IF pActValue <> 0 AND pSetValue <> 0 AND_THEN MEMCMP(pSetValue, pActValue, Len) = 0
THEN //Skip write parameter if set and actual value are equel
	state													:= state + 1;	
	setValue												:= TRUE;
ELSE
	CoEWrite(bExecute := TRUE, nIndex := Index ,nSubIndex := SubIndex , pSrcBuf := pSetValue ,cbBufLen := Len , bCompleteAccess := CompleteAccess );
	IF NOT CoEWrite.bBusy
	THEN
		IF NOT CoEWrite.bError
		THEN
			IF pActValue <> 0 THEN MEMCPY(pActValue, pSetValue, Len); END_IF	
			state											:= state + 1;
		ELSE
			Busy											:= FALSE;
			Error											:= TRUE;
			ErrorId											:= CoEWrite.nErrId;
			ErrorText										:= CONCAT('Error write parameter in state:' , TO_STRING(state * -1));
			ErrorText										:= CONCAT(ErrorText , ' Id:');
			ErrorText										:= CONCAT(ErrorText , TO_STRING(ErrorId));
			State											:= 9999;
		END_IF
		CoEWrite(bExecute := FALSE);
		setValue											:= TRUE;
	END_IF		
END_IF
END_METHOD

END_FUNCTION_BLOCK

// ---- POUs/IO/Drives/SoE/AxDriveSoE_Ax5000CommutationCalib.TcPOU
FUNCTION_BLOCK AxDriveSoE_Ax5000CommutationCalib EXTENDS FbBase
VAR CONSTANT
	STEP_COUNT											:	INT := 1;
	P150_NAMEPLATE_TYPE									:	E_AX5000_P_0150_DigitalNamePlate := E_AX5000_P_0150_DigitalNamePlate.EAX5000_P_0150_DIGITALNAMEPLATE_BECKHOFF; //1= Digital nameplate = Beckhoff
	P150_COMMUTATION_MODE_FEEDBACK						:	UINT := 1; //1= Feedback commutation offset
	
//	P150_NO_NAMEPLATE									:	UINT := 0; //0= Digital nameplate = no nameplate
//	P150_COMMUTATION_MODE_ADJUSTABLE					:	UINT := 3; //3= Adjustable mechanical offset 
END_VAR
VAR_OUTPUT CONSTANT
{attribute 'displaymode':='binary'}
	OPTION_READ_ONLY									:	BYTE  := 2#0000_0001; //Read actual commutation offset of the motor (not stored value in drive)
{attribute 'displaymode':='binary'}
	OPTION_P98_IS_EMPTY									:	BYTE  := 2#0000_0010; //Digital nameplate not initialized, skip check if entries. Select this option for first time setup
END_VAR
VAR_INPUT
	AdsAddr												: 	AMSADDR; //Terminal AMS Net Addr.	
	Channel												:	USINT;

{attribute 'displaymode':='binary'}         			
	Options												:	BYTE  := 2#0000_0000; (* Option constants are predefined, so they can accordingly be passed symbolically to the block 
																					.0 = TRUE read only 
																					*)

	
	MaxComPosDifference									:	LREAL := 15.0; //Maximal commutation position offset (Parameter P167, result of command P166)
END_VAR
VAR_IN_OUT
	axis												: AXIS_REF;
END_VAR
VAR_OUTPUT

	P0053												: AX5000_P_0053; // Configured motor type
	P0058												: AX5000_P_0058; // Mechanical commutation offset after command P166
	P0150												: AX5000_P_0150; // Feedback type form startup list
	P0167												: AX5000_P_0167; //Motor and feedback connection check parameter
	P0098												: AX5000_P_0098_beckhoff := (	
															Id_prat_1:= 1113940843,
															Id_prat_2:= 1752131174,	
														//	Name_plate_type := , 
															Version_no:=2,
															Motor_vendor:= 0, //None
															Serial_number:= 999999); //Digital nameplate
	Offset												:	LREAL; //Scaled value

	SercosErrId											: UDINT;
END_VAR
VAR
(*  Memory *****************************************************)
	lastState											: INT := 0;

(*  Timer ******************************************************)
(*  Trigger ****************************************************)

(*  Blocks *****************************************************)
	SoECommand 											: FB_SoEExecuteCommand 	:= (Timeout := t#30s);
	SoEWritePassword 									: FB_SoEWritePassword 	:= (Password :=(strData := 'AX5000', iActualSize := 128, iMaxSize := 128), Timeout := DEFAULT_ADS_TIMEOUT);
	SoEReset											: FB_SoEReset 			:= (Timeout := DEFAULT_ADS_TIMEOUT);
	SoEWrite											: FB_SoEWrite 			:= (Timeout := T#30S);
	SoERead												: FB_SoERead 			:= (Timeout := DEFAULT_ADS_TIMEOUT);
	
(*  Error ******************************************************)
(*  Dummys *****************************************************)
	{attribute 'hide' := ''}
	i,j													: INT := 0;

END_VAR

	(*********************************************************)
	
(* state machine ********************************************************)
	rtExecute(CLK := Execute);
	CASE state OF
	0 : 
		Busy 											:= FALSE;
		
		IF NOT Execute THEN
			Done 										:= FALSE;
			Error 										:= FALSE;
			ErrorID 									:= 0;
			SercosErrId									:= 0;
		END_IF
		IF rtExecute.Q THEN
			IF axis.status.ControlLoopClosed AND NOT Options.1 THEN
				Error 									:= TRUE;
				ErrorID 								:= 19266; //xis is enabled but should not be enabled for this process.

			ELSIF AdsAddr.netId[0] = 0
			THEN
 				Error 									:= TRUE;
				ErrorID 								:= 15; //Invalid AMS net id
	
			ELSIF AdsAddr.port = 0
			THEN
				Error 									:= TRUE;
				ErrorID 								:= 24; //Invalid ADS Port
						
			ELSE
				Busy									:= TRUE;	
				Done 									:= FALSE;
				Error 									:= FALSE;
				ErrorID 								:= 0;
				SercosErrId								:= 0;	
				
				Offset									:= 0.0;
				MEMSET(ADR(P0053),0,SIZEOF(P0053));
				MEMSET(ADR(P0058),0,SIZEOF(P0058));
				MEMSET(ADR(P0150),0,SIZEOF(P0150));
				MEMSET(ADR(P0167),0,SIZEOF(P0167));
				
				SoECommand(Execute := FALSE, Axis := axis);
				SoEWrite(Execute := FALSE, Axis := axis);
				SoERead(Execute := FALSE, Axis := axis);
				SoEReset(Execute := FALSE, Axis := axis);
				SoEWritePassword(Execute := FALSE, Axis := axis);
		
					
				state									:= state + STEP_COUNT;
			END_IF
		END_IF
	
	1:	(*write drive password *)
		SoEWritePassword(
			NetId:= , 
			Execute:=TRUE , 
			Timeout:= , 
			Password:= , //See declaration 
			Axis:=axis , 
			Busy=> , 
			Error=> , 
			AdsErrId=> , 
			SercosErrId=> );
	
		IF NOT SoEWritePassword.busy
		THEN
			IF SoEWritePassword.Error
			THEN
				Busy									:= FALSE;
				Error									:= TRUE;
				ErrorId									:= SoEWritePassword.AdsErrId;
				SercosErrId								:= SoEWritePassword.SercosErrId;
				state 									:= 0;
			ELSE
				
				state									:= state + STEP_COUNT;
			END_IF		
			SoEWritePassword(Execute := FALSE, Axis := axis);
		END_IF
			
	2:	(* Reset active errors *)
		SoEReset(
			NetId:= , 
			Execute:=TRUE , 
			Timeout:= , 
			Axis:=axis , 
			Busy=> , 
			Error=> , 
			AdsErrId=> , 
			SercosErrId=> );
			
		IF NOT SoEReset.Busy
		THEN
			IF SoEReset.Error
			THEN
				Busy									:= FALSE;
				Error									:= TRUE;
				ErrorId									:= SoEReset.AdsErrId;
				SercosErrId								:= SOEReset.SercosErrId;
				state 									:= 0;
			ELSE
				
				state									:= state + STEP_COUNT;
			END_IF	
			SoEReset(Execute := FALSE, Axis := axis);	
		END_IF

	3: // read configured motor type
		SoERead(
			NetId:= , 
			Idn:=P_0_IDN+53 , // IDN P-0-0053 Configured motor type
			Element:=EC_SOE_ELEMENT_VALUE , 
			pDstBuf:=ADR(P0053) , 
			BufLen:=SIZEOF(P0053) , 
			Execute:=TRUE , 
			Timeout:= , 
			Axis:=axis , 
			Busy=> , 
			Error=> , 
			AdsErrId=> , 
			SercosErrId=> , 
			Attribute=> );
			
		IF NOT SoERead.Busy
		THEN
			IF SoERead.Error
			THEN
				Busy									:= FALSE;
				Error									:= TRUE;
				ErrorId									:= SoERead.AdsErrId;
				SercosErrId								:= SoERead.SercosErrId;
				state 									:= 0;
			ELSE		
				
				state									:= state + STEP_COUNT;
			END_IF	
			SoERead(Execute := FALSE, Axis := axis);	
		END_IF
		
	4: //Read feedback type form startup list
		SoERead(
			NetId:= , 
			Idn:=P_0_IDN+150 , 
			Element:=EC_SOE_ELEMENT_VALUE , 
			pDstBuf:=ADR(P0150) , 
			BufLen:=SIZEOF(P0150) , 
			Execute:=TRUE , 
			Timeout:= , 
			Axis:=axis , 
			Busy=> , 
			Error=> , 
			AdsErrId=> , 
			SercosErrId=> , 
			Attribute=> );
			
		IF NOT SoERead.Busy
		THEN
			IF SoERead.Error
			THEN
				Busy									:= FALSE;
				Error									:= TRUE;
				ErrorId									:= SoERead.AdsErrId;
				SercosErrId								:= SoERead.SercosErrId;
				state 									:= 0;
			ELSE				
				state									:= state + STEP_COUNT;
			END_IF		
			SoERead(Execute := FALSE, Axis := axis);
		END_IF		
		
	5: (* Reserved *****************************************************)
		state											:= state + STEP_COUNT;
		
	6: //Read nameplate to check content (must be initialized) *************************
		SoERead(
			NetId:= , 
			Idn:=P_0_IDN+98 , 
			Element:=EC_SOE_ELEMENT_VALUE , 
			pDstBuf:=ADR(P0098) , 
			BufLen:=SIZEOF(P0098) , 
			Execute:=TRUE, 
			Timeout:= , 
			Axis:=axis , 
			Busy=> , 
			Error=> , 
			AdsErrId=> , 
			SercosErrId=> , 
			Attribute=> );	
		
		IF NOT SoERead.Busy
		THEN
			IF SoERead.Error
			THEN
				Busy									:= FALSE;
				Error									:= TRUE;
				ErrorId									:= SoERead.AdsErrId;
				SercosErrId								:= SoERead.SercosErrId;
				state 									:= 0;
			ELSE
				Offset									:= TO_LREAL(P0098.Position_offset) * 0.01;
				SoERead(Execute := FALSE, Axis := axis);	
				//Check parameter of P150
				IF Options.0
				THEN //Read only
					Busy								:= FALSE;
					Done								:= TRUE;
					state 								:= 0;
					
				ELSIF Options.1
				THEN //Nameplate not active, ignore current setting
					state								:= 10;	
					
				ELSIF TO_UINT(P0150.ParameterChannel.CommutationMode0) <> P150_COMMUTATION_MODE_FEEDBACK 
				THEN
					Busy								:= FALSE;
					Error								:= TRUE;
					ErrorId								:= E_AdsErr.DEVICE_INVALIDPARM;
					SercosErrId							:= 16#F749; //Feedback parameter invalid
					state 								:= 0;	
				ELSIF P0150.ParameterChannel.DigitalNamePlate <> P150_NAMEPLATE_TYPE
				THEN
					Busy								:= FALSE;
					Error								:= TRUE;
					ErrorId								:= E_AdsErr.DEVICE_INVALIDPARM;
					SercosErrId							:= 16#F749; //Invalid nameplate
					state 								:= 0;			
			
				ELSIF P0098.Name_plate_type <> P0150.ParameterChannel.DigitalNamePlate 
				THEN
					Busy								:= FALSE;
					Error								:= TRUE;
					ErrorId								:= E_AdsErr.DEVICE_INVALIDPARM;
					SercosErrId							:= 16#F803; //Unknow nameplate
					state 								:= 0;					
				
				ELSIF P0098.Position_offset = 0.0 
				THEN
					Busy								:= FALSE;
					Error								:= TRUE;
					ErrorId								:= E_AdsErr.DEVICE_INVALIDPARM;
					SercosErrId							:= 16#F742; //Invalid commutation offset
					state 								:= 0;
						
				ELSIF P0098.Feedback_typ <> P0150.FeedbackTypeString 
				THEN
					Busy								:= FALSE;
					Error								:= TRUE;
					ErrorId								:= E_AdsErr.DEVICE_INVALIDPARM;
					SercosErrId							:= 16#F708; //Feedback type invalid
					state 								:= 0;		
				ELSIF P0098.Motor_type <> P0053.Configures_motor_type 
				THEN
					Busy								:= FALSE;
					Error								:= TRUE;
					ErrorId								:= E_AdsErr.DEVICE_INVALIDPARM;
					SercosErrId							:= 16#FD09; //Motor type invalid
					state 								:= 0;				
				ELSE
					state								:= 10;	
				END_IF	
			END_IF
		END_IF
		
	10:	// Start command P-0-0160 - calibrate commutation offset ***********************************************	
		SoECommand(
			NetId:='' , 
			Idn:=P_0_IDN+160 , //command P-0-0160 = calibrate commutation offset 
			Execute:= TRUE, 
			Timeout:= , 
			Axis:=axis , 
			Busy=> , 
			Error=> , 
			AdsErrId=> , 
			SercosErrId=> );
		
		IF NOT SoECommand.Busy
		THEN
			IF SoECommand.Error
			THEN
				Busy									:= FALSE;
				Error									:= TRUE;
				ErrorId									:= SoECommand.AdsErrId;
				SercosErrId								:= SoECommand.SercosErrId;
				state 									:= 0;
			ELSE
				state									:= state + STEP_COUNT;
			END_IF		
			SoECommand(Execute := FALSE, Axis := axis);
		END_IF
	
	11: // read mechanical commutation offset result of command P160
		SoERead(
			NetId:= , 
			Idn:=P_0_IDN+58 , // IDN P-0-0167 = parameters to check commutation and rotation direction
			Element:=EC_SOE_ELEMENT_VALUE , 
			pDstBuf:=ADR(P0058) , 
			BufLen:=SIZEOF(P0058) , 
			Execute:= TRUE , 
			Timeout:= , 
			Axis:=axis , 
			Busy=> , 
			Error=> , 
			AdsErrId=> , 
			SercosErrId=> , 
			Attribute=> );	
		
		IF NOT SoERead.Busy
		THEN
			IF SoERead.Error
			THEN
				Busy									:= FALSE;
				Error									:= TRUE;
				ErrorId									:= SoERead.AdsErrId;
				SercosErrId								:= SoERead.SercosErrId;
				state 									:= 0;
			ELSE
				//Init nameplate information - see also declaration
				P0098.Motor_type						:= P0053.Configures_motor_type;
				P0098.Feedback_typ						:= P0150.FeedbackTypeString;	
				P0098.Name_plate_type					:= P0150.ParameterChannel.DigitalNamePlate;
				P0098.Position_offset					:= P0058.Mechanical_commutation_offset;
				Offset									:= TO_LREAL(P0058.Mechanical_commutation_offset) * 0.01;		
	
				state									:= state + STEP_COUNT;
			END_IF	
			SoERead(Execute := FALSE, Axis := axis);	
		END_IF
		
	12: // Start command P-0-0166 - Motor and feedback connection check 
		SoECommand(
			NetId:='' , 
			Idn:=P_0_IDN+166 , //command P-0-0166 = motor and feedback connection check 
			Execute:= TRUE, 
			Timeout:= , 
			Axis:=axis , 
			Busy=> , 
			Error=> , 
			AdsErrId=> , 
			SercosErrId=> );
		
		IF NOT SoECommand.Busy
		THEN
			IF SoECommand.Error
			THEN
				Busy									:= FALSE;
				Error									:= TRUE;
				ErrorId									:= SoECommand.AdsErrId;
				SercosErrId								:= SoECommand.SercosErrId;
				state 									:= 0;
			ELSE
				
				state									:= state + STEP_COUNT;
			END_IF		
			SoECommand(Execute := FALSE, Axis := axis);
		END_IF
	
	13: // read P-0-0167 read connection check results
		SoERead(
			NetId:= , 
			Idn:=P_0_IDN+167 , // IDN P-0-0167 = parameters to check commutation and rotation direction
			Element:=EC_SOE_ELEMENT_VALUE , 
			pDstBuf:=ADR(P0167) , 
			BufLen:=SIZEOF(P0167) , 
			Execute:= TRUE , 
			Timeout:= , 
			Axis:=axis , 
			Busy=> , 
			Error=> , 
			AdsErrId=> , 
			SercosErrId=> , 
			Attribute=> );
				
		IF NOT SoERead.Busy
		THEN
			IF SoERead.Error
			THEN
				Busy									:= FALSE;
				Error									:= TRUE;
				ErrorId									:= SoERead.AdsErrId;
				SercosErrId								:= SoERead.SercosErrId;
				state 									:= 0;
			ELSE				
				IF P0167.EqualDirektions <> 1
					OR
					TO_LREAL(P0167.Commutation_position_difference) * 0.01 > MaxComPosDifference 
					AND TO_LREAL(P0167.Commutation_position_difference) * 0.01 < 360.0 - MaxComPosDifference
				THEN
					Busy								:= FALSE;
					Error								:= TRUE;
					ErrorId								:= E_AdsErr.DEVICE_INVALIDPARM;
					SercosErrId							:= 16#F702; //Feedback position invalid
					state 								:= 0;
				ELSE                                	
					state								:= state + STEP_COUNT;
				END_IF
			END_IF		
			SoERead(Execute := FALSE, Axis := axis);
		END_IF
		
	14:	// Write digital motor plate with commutation offset
		SoEWrite(
			NetId:= , 
			Idn:=P_0_IDN+98, // P0-0-0098 = digital motor plate 
			Element:=EC_SOE_ELEMENT_VALUE , 
			pSrcBuf:=ADR(P0098) ,
			BufLen:=SIZEOF(P0098) ,
			Execute:=TRUE,
			Timeout:= , 
			Password:= SoEWritePassword.Password, 
			Axis:=axis , 
			Busy=> , 
			Error=> , 
			AdsErrId=> , 
			SercosErrId=> );
			
		IF NOT SoEWrite.Busy
		THEN
			IF SoEWrite.Error
			THEN
				Busy									:= FALSE;
				Error									:= TRUE;
				ErrorId									:= SoEWrite.AdsErrId;
				SercosErrId								:= SoEWrite.SercosErrId;
				state 									:= 0;
			ELSE
				
				state									:= state + STEP_COUNT;
			END_IF	
			SoEWrite(Execute := FALSE, Axis := axis);	
		END_IF

	15: // Command P-0-0162 - Save digital name plate
		SoECommand(
			NetId:= , 
			Idn:=P_0_IDN+162 , //save digital name plate 
			Execute:=TRUE , 
			Timeout:= , 
			Axis:=axis , 
			Busy=> , 
			Error=> , 
			AdsErrId=> , 
			SercosErrId=> );
	
		IF NOT SoECommand.Busy
		THEN
			IF SoECommand.Error
			THEN
				Busy									:= FALSE;
				Error									:= TRUE;
				ErrorId									:= SoECommand.AdsErrId;
				SercosErrId								:= SoECommand.SercosErrId;
				state 									:= 0;
			ELSE
				
				state									:= state + STEP_COUNT;
			END_IF		
			SoECommand(Execute := FALSE, Axis := axis);
		END_IF

	16: // Write digital motor plate with commutation offset again
		SoEWrite(
			NetId:= , 
			Idn:=P_0_IDN+98 , 
			Element:=EC_SOE_ELEMENT_VALUE , 
			pSrcBuf:=ADR(P0098) ,
			BufLen:=SIZEOF(P0098) ,
			Execute:= TRUE,
			Timeout:= , 
			Password:=SoEWritePassword.Password  , 
			Axis:=axis , 
			Busy=> , 
			Error=> , 
			AdsErrId=> , 
			SercosErrId=> );
				
		IF NOT SoEWrite.Busy
		THEN
			IF SoEWrite.Error
			THEN
				Busy									:= FALSE;
				Error									:= TRUE;
				ErrorId									:= SoEWrite.AdsErrId;
				SercosErrId								:= SoEWrite.SercosErrId;
				state 									:= 0;
			ELSE
				
				state									:= state + STEP_COUNT;
			END_IF	
			SoEWrite(Execute := FALSE, Axis := axis);	
		END_IF

	17: //Start command P-0-0161 - Save commutation offset in feedback 1
		SoECommand(
			NetId:= , 
			Idn:=P_0_IDN+161 , //save commutation offset 
			Execute:=TRUE , 
			Timeout:= , 
			Axis:=axis , 
			Busy=> , 
			Error=> , 
			AdsErrId=> , 
			SercosErrId=> );
		
		IF NOT SoECommand.Busy
		THEN
			IF SoEWrite.Error
			THEN
				Busy									:= FALSE;
				Error									:= TRUE;
				ErrorId									:= SoEWrite.AdsErrId;
				SercosErrId								:= SoEWrite.SercosErrId;
				state 									:= 0;
			ELSE
				Busy									:= FALSE;
				Done									:= TRUE;
				state 									:= 0;					
			END_IF		
			SoECommand(Execute := FALSE, Axis := axis);
		END_IF
	
	ELSE
		;
	END_CASE

(* Record last state ******************************************)
IF state <> lastState AND state <> 0 AND NOT Error
THEN 
	lastState											:= state;
END_IF

(*************************************************************)

{attribute 'monitoring' := 'call'}
PROPERTY PUBLIC optP98IsEmpty : BOOL
GET
optP98IsEmpty := Options.1;
END_GET
SET
Options.1 := optP98IsEmpty;
END_SET
END_PROPERTY

{attribute 'monitoring' := 'call'}
PROPERTY PUBLIC optReadOnly : BOOL
GET
optReadOnly := Options.0;
END_GET
SET
Options.0 := optReadOnly;
END_SET
END_PROPERTY

END_FUNCTION_BLOCK

// ---- POUs/IO/Drives/SoE/AxDriveSoE_Ax5000SwitchParamSet.TcPOU
FUNCTION_BLOCK AxDriveSoE_Ax5000SwitchParamSet EXTENDS FbBase
VAR_INPUT
	rAxis													:	REFERENCE TO AXIS_REF := 0; 	// Axis Ref
	TimeOut													:	TIME := DEFAULT_ADS_TIMEOUT;	// Timeout time
	NewParamSet												:	INT;							// Value for new parameterset
END_VAR
VAR_IN_OUT	
(* important for function *)	
	AdsAddr													:	AMSADDR;						// AdsAddr of AX5000
	Channel													:	USINT;                          // Drive channel number
END_VAR
VAR_OUTPUT
	ErrorText												:	T_MaxString;					// Error Text
	ActParamSet												:	INT := -1; 						// Value of active parameter set
END_VAR
VAR
(* Memory **********************************************************)
	StartSwitchParamSet										:	INT := 0;
	
	CountError												:	USINT;
(* Timer ***********************************************************)
	TimerWait												:	TON;
	TimerTimeOut											:	TON;
	
(* Functionsblocks *************************************************)

	SoEWrite												:	FB_SoEWrite_ByDriveRef	:= (tTimeOut := DEFAULT_ADS_TIMEOUT);
	SoERead													:	FB_SoERead_ByDriveRef	:= (tTimeOut := DEFAULT_ADS_TIMEOUT);
(*******************************************************************)
END_VAR
VAR CONSTANT
	ST_IDLE													:	INT := 0;
	ST_REFRESH												:	INT := 10;
	ST_PRESELECT											:	INT := 100;
	ST_DISABLED												:	INT := 110;
	ST_RESETEXECUTE											:	INT := 120;
	ST_SETPARAM												:	INT := 130;
	ST_WAIT													:	INT := 140;
	ST_ERROR												:	INT := 998;
	ST_RESET												:	INT := 999;
	
	ERR_REFRESH												:	UDINT := 1;
	ERR_PRESELECT											:	UDINT := 2;
	ERR_TIMEOUT_DISABLED									:	UDINT := 3;
	ERR_RESETEXECUTE										:	UDINT := 4;
	ERR_EXECUTE												:	UDINT := 5;
	
	PT_WAIT_TIME											:	TIME := T#20MS;
END_VAR

(* abort function-call if the reference is invalid *****************)
	IF NOT __ISVALIDREF(rAxis) THEN
		Busy												:= NOT Error;
		Error												:= TRUE;
		ErrorId												:= 16#4B30;
		ErrorText											:= 'Referenz rAxis invalid (0)';
		RETURN;
	END_IF

(* Init drive ref **************************************************)
	IF AdsAddr.port <> SoERead.stDriveRef.nSlaveAddr
	THEN
		SoERead.stDriveRef.sNetId							:= F_CreateAmsNetId(AdsAddr.netId);
		SoERead.stDriveRef.nSlaveAddr						:= AdsAddr.port;
		SoERead.stDriveRef.nDriveNo							:= Channel;
		
		SoEWrite.stDriveRef									:= SoERead.stDriveRef;
	END_IF
(* Trigger Execute *************************************************)
	rtExecute(CLK := Execute);
	
(* switch parameter set ********************************************)
	CASE State OF
	ST_IDLE:			// wait for command
	(* Get actual parameter set after restart *)
		IF ActParamSet < 0 
		THEN
			State											:= ST_REFRESH;
	(* Start switch parameter set *)
		ELSIF rtExecute.Q
		THEN
			setNewParam(NewParamSet);
		ELSIF NOT Execute
		THEN
			Error											:= FALSE;
			Done											:= FALSE;
			Busy											:= TRUE;
			ErrorId											:= 0;
			ErrorTExt										:= '';
		END_IF
		
	ST_REFRESH: 		// Refresh ActParamSet Variable
		IF NOT SoERead.bBusy
			AND SoERead.bExecute
		THEN
			State											:= SEL(SoERead.bError, ST_IDLE, ST_ERROR);
			Done											:= State = ST_IDLE;
			Error											:= State = ST_ERROR;	
			ErrorID											:= SEL(SoERead.bError, 0, ERR_REFRESH);
			ErrorText										:= SEL(SoERead.bError, '', 'Fehler beim Aktualisieren des aktuellen Parametersatzes');
		END_IF
		
		SoERead(
			stDriveRef	:= ,  //See init for drive ref
			nIdn		:= S_0_IDN + 254,
			nElement	:= EC_SOE_ELEMENT_VALUE (* 16#40*),
			pDstBuf		:= ADR(ActParamSet),
			cbBufLen	:= SIZEOF(ActParamSet),
			bExecute	:= State = ST_REFRESH,
			tTimeout	:= ,
			bBusy		=> ,
			bError		=> ,
			iAdsErrId	=> ,
			iSercosErrId=> ,
			dwAttribute	=> );
			
		ST_PRESELECT:		// Set New param value in drive preselection
			IF NewParamSet = ActParamSet
			THEN
				State										:= ST_IDLE;
			ELSIF NOT SoEWrite.bBusy
				AND SoEWrite.bExecute
			THEN
				State										:= SEL(SoEWrite.bError, ST_DISABLED, ST_ERROR);
				ErrorID										:= SEL(SoERead.bError, 0, ERR_PRESELECT);
				ErrorText									:= SEL(SoERead.bError, '', 'Fehler beim Schreiben der Vorwahl');
			END_IF
			
			SoEWrite(
				stDriveRef	:= ,  //See init for drive ref
				nIdn		:= S_0_IDN + 217,
				nElement	:= EC_SOE_ELEMENT_VALUE (* 16#40*),
				pSrcBuf		:= ADR(NewParamSet),
				cbBufLen	:= SIZEOF(NewParamSet),
				bExecute	:= State = ST_PRESELECT,
				tTimeout	:= ,
				bBusy		=> ,
				bError		=> ,
				iAdsErrId	=> ,
				iSercosErrId=> );
				
		ST_DISABLED:		// check if axis is disabled
			TimerTimeOut(IN := NOT rAxis.Status.Disabled, PT := TimeOut);
			IF TimerTimeOut.Q THEN
				TimerTimeOut(IN := FALSE);
				State											:= ST_ERROR;
				ErrorID											:= SEL(SoERead.bError, 0, ERR_TIMEOUT_DISABLED);
				ErrorText										:= SEL(SoERead.bError, '', 'Achse ist nicht deaktiviert');
			ELSIF rAxis.Status.Disabled THEN
				TimerTimeOut(IN := FALSE);
				State											:= ST_RESETEXECUTE;
			END_IF
		
		ST_RESETEXECUTE:	// reset the execute command in drive	
			StartSwitchParamSet									:= 0;
			IF NOT SoEWrite.bBusy
				AND SoEWrite.bExecute
			THEN
				State											:= SEL(SoEWrite.bError, ST_SETPARAM, ST_ERROR);
				ErrorID											:= SEL(SoERead.bError, 0, ERR_RESETEXECUTE);
				ErrorText										:= SEL(SoERead.bError, '', 'Fehler beim Zurücksetzen des Ausführungskomamando');
			END_IF
			SoEWrite(
				stDriveRef	:= ,  //See init for drive ref
				nIdn		:= S_0_IDN + 216,
				nElement	:= EC_SOE_ELEMENT_VALUE (* 16#40*),
				pSrcBuf		:= ADR(StartSwitchParamSet),
				cbBufLen	:= SIZEOF(StartSwitchParamSet),
				bExecute	:= State = ST_RESETEXECUTE,
				tTimeout	:= ,
				bBusy		=> ,
				bError		=> ,
				iAdsErrId	=> ,
				iSercosErrId=> );		
				
		ST_SETPARAM:		// Execute switch parameter set
			StartSwitchParamSet								:= 3;
			IF NOT SoEWrite.bBusy
				AND SoEWrite.bExecute
			THEN
				State										:= SEL(SoEWrite.bError, ST_WAIT, ST_ERROR);
				ErrorID										:= SEL(SoERead.bError, 0, ERR_EXECUTE);
				ErrorText									:= SEL(SoERead.bError, '', 'Fehler beim Setzen des Ausführungskommandos');
			END_IF
			SoEWrite(
				stDriveRef	:= ,  //See init for drive ref
				nIdn		:= S_0_IDN + 216,
				nElement	:= EC_SOE_ELEMENT_VALUE (* 16#40*),
				pSrcBuf		:= ADR(StartSwitchParamSet),
				cbBufLen	:= SIZEOF(StartSwitchParamSet),
				bExecute	:= State = ST_SETPARAM,
				tTimeout	:= ,
				bBusy		=> ,
				bError		=> ,
				iAdsErrId	=> ,
				iSercosErrId=> );
				
		ST_WAIT:			// wait a short time while the drive works with the command
			TimerWait(IN := TRUE, pt := PT_WAIT_TIME);
			IF TimerWait.Q THEN
				TimerWait(IN := FALSE);
				State										:= ST_REFRESH;
			END_IF
			
		ST_ERROR:			// wait till Error is quit
			IF TRUE
			THEN
				State										:= ST_RESET;
			END_IF
			
		ST_RESET:			// Reset Error			
			State											:= ST_IDLE;
			SoEWrite(
				stDriveRef	:= ,  //See init for drive ref
				nIdn		:= S_0_IDN + 216,
				nElement	:= EC_SOE_ELEMENT_VALUE (* 16#40*),
				pSrcBuf		:= ADR(StartSwitchParamSet),
				cbBufLen	:= SIZEOF(StartSwitchParamSet),
				bExecute	:= FALSE,
				tTimeout	:= ,
				bBusy		=> ,
				bError		=> ,
				iAdsErrId	=> ,
				iSercosErrId=> );
			SoERead(
				stDriveRef	:= ,  //See init for drive ref
				nIdn		:= S_0_IDN + 254,
				nElement	:= EC_SOE_ELEMENT_VALUE (* 16#40*),
				pDstBuf		:= ADR(ActParamSet),
				cbBufLen	:= SIZEOF(ActParamSet),
				bExecute	:= FALSE,
				tTimeout	:= ,
				bBusy		=> ,
				bError		=> ,
				iAdsErrId	=> ,
				iSercosErrId=> ,
				dwAttribute	=> );
	END_CASE
	Busy													:= State <> ST_IDLE ;
(*******************************************************************)

METHOD setNewParam : BOOL	// Result = Busy
VAR_INPUT
	ParamNo					:	INT;
END_VAR

	IF ParamNo <> ActParamSet
		AND State = ST_IDLE
	THEN
		Error											:= FALSE;
		Done											:= FALSE;
		Busy											:= TRUE;
		ErrorId											:= 0;
		ErrorTExt										:= '';
		NewParamSet 									:= ParamNo;
		TimerWait(IN := FALSE);
		TimerTimeOut(IN := FALSE);
		State											:= ST_PRESELECT;
	END_IF
	
	SetNewParam											:= State <> ST_IDLE;
END_METHOD

END_FUNCTION_BLOCK

// ---- POUs/IO/EL-EP/EL1262_Base.TcPOU
FUNCTION_BLOCK EL1262_Base
VAR_INPUT
END_VAR
VAR_OUTPUT
	Input										AT %I*		:	BOOL;
{attribute 'displaymode':='binary'}
	Status										AT %I*		:	USINT;
	TimeLatchPos								AT %I*		:	T_DCTIME64;
	TimeLatchNeg								AT %I*		:	T_DCTIME64;
END_VAR
VAR
END_VAR

END_FUNCTION_BLOCK

// ---- POUs/IO/EL-EP/EL9x/EL9501.TcPOU
{attribute 'no_check'}
FUNCTION_BLOCK EL9501 EXTENDS EcSlaveInfoDataExt
VAR_INPUT
	SetVoltage					AT %Q*		:	REAL; // 0.0 - 20.0 [V]
END_VAR                 					 	
VAR_OUTPUT    
	{attribute 'displaymode':='binary'}             	
	Status						AT  %I*		:	WORD; // Terminal status (2 bytes)
          					 	
	Voltage								 	: 	AnalogInREAL ; 
	Current								 	: 	AnalogInREAL;
END_VAR                                 
VAR                                     

END_VAR

	(* EL9501 Power supply terminal	 0-20V	*)
	(****************************************)
	SUPER^();
	
(* Work objects *****************************)
	Voltage();
	Current();

(********************************************)

{attribute 'monitoring' := 'call'}
PROPERTY PUBLIC error : BOOL
GET
Error				:= Status.6 OR Voltage.Error OR Current.Error;
END_GET
END_PROPERTY

METHOD PUBLIC off : BOOL
VAR_INPUT
END_VAR
Off := CAM(SetVoltage, Voltage.Q, 0.01);
END_METHOD

{attribute 'monitoring' := 'call'}
PROPERTY PUBLIC overload : BOOL
GET
Overload 			:= Status.1;
END_GET
END_PROPERTY

{attribute 'monitoring' := 'call'}
PROPERTY PUBLIC overrange : BOOL
GET
Overrange 			:= Status.3;
END_GET
END_PROPERTY

{attribute 'monitoring' := 'call'}
PROPERTY PUBLIC underrange : BOOL
GET
Underrange 			:= Status.2;
END_GET
END_PROPERTY

{attribute 'monitoring' := 'call'}
PROPERTY PUBLIC warning : BOOL
GET
Warning 			:= Status.5;
END_GET
END_PROPERTY

END_FUNCTION_BLOCK

// ---- POUs/IO/_EcSlaveInfoDataIO/EcSlaveInfoDataExt.TcPOU
{attribute 'no_check'}
{attribute 'reflection'} 
FUNCTION_BLOCK EcSlaveInfoDataExt Extends EcSlaveInfoData
VAR_INPUT
END_VAR                         					
VAR_OUTPUT                      					
	AmsNetIdStr												: T_AmsNetId; //AMS NetID string
	EcMasterDevId									AT %I*	: UINT; 	// Link to EtherCAT Master "DevId" under InfoData 
	DevName													:	STRING(30) := ''; //Slave device name as give in IO tree				
	{attribute 'instance-path'} 
    {attribute 'noinit'} 
    InstancePath 											: STRING; 	
END_VAR
VAR
	IOF_GetBoxNameByAddr									:	IOF_GetBoxNameByAddr := (NETID := '', TMOUT := DEFAULT_ADS_TIMEOUT);
	_Init_													: BOOL;
END_VAR

(* Get device name by address and master device id								*)
(********************************************************************************)

(* Get name *********************************************************************)
IF NOT _Init_
THEN 	
	IF NOT IOF_GetBoxNameByAddr.START
	THEN
		IF AdsAddr.port = 0 
		THEN
			adsLogError('AdsAddr.port invalid: %s', InstancePath);
		END_IF
		IF EcMasterDevId = 0 
		THEN
			adsLogError('EcMasterDevId invalid: %s', InstancePath);
		END_IF
			
		IF AdsAddr.port > 0 AND EcMasterDevId > 0
		THEN
			IOF_GetBoxNameByAddr.START						:= TRUE;
			AmsNetIdStr										:= F_CreateAmsNetId(nIds := AdsAddr.netId);
		END_IF		
	END_IF
	
	IOF_GetBoxNameByAddr(
		NETID		:=  , (* Local *)
		DEVICEID	:= TO_UDINT(EcMasterDevId) ,
		BOXADDR		:= AdsAddr.port ,
		START		:= ,
		TMOUT		:= ,
		BOXNAME		=> DevName);
	IF NOT IOF_GetBoxNameByAddr.BUSY 
	THEN
		IF IOF_GetBoxNameByAddr.ERR 
		THEN
			adsLogError(CONCAT(CONCAT('ADS Error ', DWORD_TO_HEXSTR(IOF_GetBoxNameByAddr.ERRID,4,FALSE)),' reading BoxName of EtherCAT Device: %s'), InstancePath);
		END_IF
		IOF_GetBoxNameByAddr(START:= FALSE);
		_Init_												:= TRUE;
	END_IF
END_IF
(********************************************************************************)

END_FUNCTION_BLOCK

// ---- POUs/IO/EL-EP/EL3356.TcPOU
{attribute 'no_check'}
//EL3356 load cell analysis (resistor bridge) process image
//Mode of operation = Standard (Real or INT32)
FUNCTION_BLOCK EL3356 EXTENDS EcSlaveInfoDataExt
VAR_INPUT
//RMB Control
	StartCalib										AT  %Q* : 	BOOL; 
	DisableCalib									AT  %Q* : 	BOOL;
	InputFreeze										AT  %Q* : 	BOOL;
	SampleMode										AT  %Q* : 	BOOL; //1=High speed and low latency / only on EL3356-0010
	Tara											AT  %Q* : 	BOOL;				
END_VAR                     			    					
VAR_OUTPUT                      					
//RMB Status
	Overrange										AT  %I*	:	BOOL;
	DataInvalid										AT  %I*	:	BOOL;
	Error											AT  %I*	:	BOOL;
	CalibInProgress									AT  %I*	:	BOOL;
	SteadyState										AT  %I*	:	BOOL;
	SyncError										AT  %I*	:	BOOL;
	TxPDOToggle										AT  %I* : 	BOOL;
	
//RMB Value
	InReal											AT  %I* : 	REAL; //RMP Value Real 32		
	InInt32											AT  %I* : 	DINT; //RMB Value INT32
END_VAR
VAR
END_VAR

(* EL3356 IOs											             	 		*)
(********************************************************************************)

(* ******************************************************************************)
	Super^();
(********************************************************************************)

{attribute 'monitoring' := 'call'}
PROPERTY PUBLIC inError : BOOL
GET
inError													:= Error OR SyncError OR WcState OR InfoDataState <> Tc2_EtherCAT.EC_DEVICE_STATE_OP;
END_GET
END_PROPERTY

{attribute 'monitoring' := 'call'}
PROPERTY PUBLIC Q : LREAL
GET
IF InInt32 <> 0
THEN
	Q 														:= TO_LREAL(InInt32);
ELSE
	Q 														:= TO_LREAL(InReal);
END_IF
END_GET
END_PROPERTY

{attribute 'monitoring' := 'call'}
PROPERTY Q_GramToNewton : LREAL
GET
Q_GramToNewton := GF_TO_N(Q);
END_GET
END_PROPERTY

{attribute 'monitoring' := 'call'}
PROPERTY Q_NewtonToGram : LREAL
GET
Q_NewtonToGram := N_TO_GF(Q);
END_GET
END_PROPERTY

END_FUNCTION_BLOCK

// ---- POUs/_Miscellaneous/Conversions/GF_TO_N.TcPOU
{attribute 'no_check'}
//Gram-force to newton
FUNCTION GF_TO_N : LREAL
VAR_INPUT
	GF				:	LREAL;
END_VAR
VAR
END_VAR
(*
Gram-force to newton (gf to N):
Fn = Fgf ×0.00980665
Example:
If gf = 156 then N = 1.5298374N

Newton to gram-force (N to gf):
Fgf = Fn / 0.00980665
*)

GF_TO_N := GF * 0.00980664999999998 ;

END_FUNCTION

// ---- POUs/_Miscellaneous/Conversions/N_TO_GF.TcPOU
{attribute 'no_check'}
//Newton to Gram-force
FUNCTION N_TO_GF : LREAL
VAR_INPUT
	FN				:	LREAL;
END_VAR
VAR
END_VAR
(*
Gram-force to newton (gf to N):
Fn = Fgf ×0.00980665
Example:
If gf = 156 then N = 1.5298374N

Newton to gram-force (N to gf):
Fgf = Fn / 0.00980665
*)

N_TO_GF := FN / 0.00980664999999998;

END_FUNCTION

// ---- POUs/IO/EL-EP/EP92xxPwrBox/EP9214_CHANNEL.TcPOU
{attribute 'no_check'}
FUNCTION_BLOCK EP9214_CHANNEL
VAR_INPUT
	EnableUs									AT  %Q* 	: 	BOOL := TRUE; 	//switches system voltage on with a rising edge
	EnableUp									AT  %Q* 	: 	BOOL := TRUE; 	//switches peripheral voltage on with a rising edge
	ResetTrigUs	                                AT  %Q* 	: 	BOOL := FALSE;  //resets system voltage with a rising edge                    
	ResetTrigUp                                 AT  %Q* 	: 	BOOL := FALSE;	//resets peripheral voltage with a rising edge                                                                                           
END_VAR     								                          
VAR_OUTPUT  								                          
	ErrorUs										AT  %I* 	: 	BOOL := FALSE;	//TRUE when system voltage error occurs 
	ErrorUp										AT  %I* 	: 	BOOL := FALSE; 	//TRUE when peripheral voltage error occurs 
	WarningUs									AT  %I* 	: 	BOOL := FALSE; 	//TRUE when system voltage warning occurs 
	WarningUp									AT  %I* 	: 	BOOL := FALSE; 	//TRUE when peripheral voltage warning occurs 
	StatusUs									AT  %I* 	: 	BOOL := FALSE; 	//TRUE when system voltage is on
	StatusUp									AT  %I* 	: 	BOOL := FALSE; 	//TRUE when peripheral voltage is on 
	ChannelError								AT  %I* 	: 	BOOL := FALSE; 	//TRUE when channel error occurs 
	SyncError									AT  %I* 	: 	BOOL := FALSE; 	//TRUE when synchronization error occurs 
	TxPDOState									AT  %I* 	: 	BOOL := FALSE; 
	TxPDOToggle									AT  %I* 	: 	BOOL := FALSE; 
END_VAR     								
VAR
END_VAR

;

END_FUNCTION_BLOCK

// ---- POUs/IO/Fuse.TcPOU
{attribute 'no_check'}
//Fuse/Circuit breaker 
FUNCTION_BLOCK Fuse
VAR_INPUT
	Force													:	BOOL := FALSE;	//simulates Input
	Invert													:	BOOL := FALSE; 	//inverts the Hardware Input
	ResetTrig												:	BOOL := TRUE;	//Resets error with rising edge 
END_VAR     								
VAR_OUTPUT  								
	Q														:	BOOL;			//output
	Event													:	BOOL;			//TRUE when state is abnormal and error is not reset 
	In											AT  %I* 	: 	BOOL := TRUE;	//Hardware Input
END_VAR     								
VAR
END_VAR

(* signallocked Input-FB (MSS,Sicherung)				*)
(********************************************************)

(************************************)
IF NOT (In OR Force) XOR Invert
THEN
	Event													:= TRUE;
	Q														:= Invert;
ELSIF Event                         						
THEN                                						
	Event 													:= NOT ResetTrig;
ELSE                                						
	Q														:= Not Invert;
END_IF

(************************************)

METHOD PUBLIC reset : BOOL
VAR_INPUT
END_VAR
Event := FALSE;
reset := TRUE;
END_METHOD

END_FUNCTION_BLOCK

// ---- POUs/IO/InOut.TcPOU
{attribute 'no_check'}
FUNCTION_BLOCK InOut 
VAR_INPUT
	Q												AT  %Q*	:	BOOL; //Link to hardware output
END_VAR             								
VAR_OUTPUT          								
	In												AT  %I*	:	BOOL; //Link to hardware input
END_VAR
VAR
END_VAR

;

END_FUNCTION_BLOCK

// ---- POUs/IO/Motors/IOMotor.TcPOU
{attribute 'no_check'}
FUNCTION_BLOCK IOMotor IMPLEMENTS I_ActuatorOnOff
VAR_INPUT
	ResetTrig												:	BOOL := TRUE; //Confirm error
	start													:	BOOL;
	Feed													:	BOOL;
	ProtSwitchOK											: 	FUSE;
END_VAR                 							
VAR_OUTPUT
{attribute 'displaymode':='binary'}
	Status													:	BYTE;              							
	Q_Contactor										AT  %Q* :	BOOL; //Hardware output for main contactor to start motor	
	Busy													:	BOOL;
	Error													:	BOOL;
END_VAR                 							
VAR (* IO Internal *)   							

                        	
END_VAR                 	
VAR                     	
END_VAR

(* Com Motor IO 					 		V2.2		*)
(********************************************************)

(* Protection Switch *****************************************)
	IF ResetTrig THEN reset(); END_IF

	ProtSwitchOK();

(* Enable ****************************************************)
	IF Start THEN
		switchOn();
	ELSE
		switchOff();
	END_IF
	
(* HMI status *********************************************)
	_writeStatus();
	
(********************************************************)

METHOD PROTECTED _writeStatus : BOOL
VAR_INPUT
END_VAR
	
(* HmiStatus **************************************************)
	Status.0												:= NOT Q_Contactor;
	Status.1												:= Q_Contactor;
	Status.2												:= FALSE;
	Status.3												:= FALSE;
	Status.4												:= FALSE;
	Status.5												:= Feed ;
	Status.6												:= NOT Error;
	Status.7												:= Error;

	(* Result *)
	_writeStatus											:= TRUE;
    												
(**************************************************************)
END_METHOD

METHOD enable : BOOL //Result value = successful execution of desired action 
VAR_INPUT
	IN							:	BOOL; //TRUE = Enable Pos/FWD/Up/Open/Left/Work FALSE = Opposite
END_VAR
IF in
THEN
	enable := switchOn();
ELSE
	enable := switchOff();
END_IF
END_METHOD

{attribute 'monitoring' := 'call'}
PROPERTY public inError : bool
GET
inError := Error;
END_GET
END_PROPERTY

{attribute 'monitoring' := 'call'}
PROPERTY public isBusy : bool
GET
isBusy := Busy;
END_GET
END_PROPERTY

{attribute 'monitoring' := 'call'}
PROPERTY public isOff : BOOL
GET
isOff := not Q_Contactor;
END_GET
END_PROPERTY

{attribute 'monitoring' := 'call'}
PROPERTY public isOn : BOOL
GET
isOn := Q_Contactor;
END_GET
END_PROPERTY

{attribute 'monitoring' := 'call'}
PROPERTY noFeed : BOOL
GET
noFeed := NOT Feed;
END_GET
END_PROPERTY

{attribute 'monitoring' := 'call'}
PROPERTY ok : bool
GET
ok := isBusy;
END_GET
END_PROPERTY

METHOD PUBLIC reset : bool
VAR_INPUT
END_VAR
Error									:= FALSE;
reset									:= ProtSwitchOK.reset();
END_METHOD

METHOD public switchOff : BOOL  //True if motor is switched off
VAR_INPUT
END_VAR
Start														:= FALSE;
Q_Contactor 												:= FALSE;
Busy														:= FALSE;
Error														:= NOT ProtSwitchOK.Q;
switchOff													:= TRUE;
END_METHOD

METHOD public switchOn : BOOL  //True if motor is switched on
VAR_INPUT
END_VAR
Start														:= TRUE;
Q_Contactor		 											:= ProtSwitchOK.Q AND Feed;
switchOn													:= Q_Contactor;
Busy														:= switchOn;
Error														:= NOT ProtSwitchOK.Q;
END_METHOD

END_FUNCTION_BLOCK

// ---- POUs/IpcDiag/MDP/InfoModuls/MDP_Mainboard.TcPOU
{attribute 'no_check'}
FUNCTION_BLOCK MDP_Mainboard  EXTENDS FbBase
VAR_OUTPUT CONSTANT
	MIN_VOLTAGE												:	INT := 1;
	MAX_VOLTAGE												:	INT := 20;

(* Voltage Location *)
 	VLOC_UNKNOWN											:	INT := 0;
	VLOC_OTHER												:	INT := 1;
 	VLOC_PROCESSOR											:	INT := 2;
 	VLOC_DISK												:	INT := 3;
 	VLOC_SYSTEM_MANAGEMENT_MODULE							:	INT := 4;
 	VLOC_MOTHERBOARD										:	INT := 5;
 	VLOC_MEMORY_MODULE										:	INT := 6;
 	VLOC_POWER_SUPPLY										:	INT := 7;
 	VLOC_ADDIN_CARD											:	INT := 8;
 	VLOC_FRONT_PANEL_BOARD									:	INT := 9;
 	VLOC_BACK_PANEL_BOARD									:	INT := 10;
 	VLOC_PERIPHERIE											:	INT := 11;
 	VLOC_CHASSIS											:	INT := 12;
 	VLOC_BATTERY											:	INT := 13;
 	VLOC_UPS												:	INT := 14;
	VLOC_GRAFFIC_BOARD										:	INT := 15;
 	VLOC_SUPERIO											:	INT := 16;
	VLOC_CHIPSET											:	INT := 17;
END_VAR                             						
VAR_INPUT                           						
	AmsNetId												: 	T_AmsNetId := '';				//AmsNetId as text
	Timeout													:	TIME := DEFAULT_ADS_TIMEOUT;	//Ads timeout
END_VAR
VAR_OUTPUT
	MB_Type													:	STRING(20);	//Type of Mainboard
	SerielNo												:	STRING(20);	//Serial number of Mainboard
	ProdDate												:	STRING(20);	//Production date of Mainboard
	BootCount												:	UDINT;		//total number of boots
	OpTime													:	UDINT; 		//Operating Time
	MinBoardTemp											:	DINT;		//minimum board temperature
	MaxBoardTemp											:	DINT;		//maximum board temperature
	MinInputVolt											:	DINT;		//minimum board input voltage
	MaxInputVolt											:	DINT;		//maximum board input voltage
	MB_Temp													:	INT;		//current board temperature
	IPC_SerielNo											:	STRING(20);	//industrial PC serial number
                        									
	VoltLocation											:  	ARRAY[MIN_VOLTAGE..MAX_VOLTAGE] OF INT;	//voltage location
	VoltageValue											:	ARRAY[MIN_VOLTAGE..MAX_VOLTAGE] OF INT;	//voltage value
	VoltageNominal											:	ARRAY[MIN_VOLTAGE..MAX_VOLTAGE] OF INT;	//nominal voltage
	VoltCount												:	INT; 		//number of measuring points
	ErrorGrp												:	E_MDP_ErrGroup := eMDP_Err_NoError;

END_VAR                 									
VAR                     									
	idx														:	INT := 1;
	MDP_ScanModules											:	FB_MDP_ScanModules := ( nModuleType 	:= eMDP_ModT_Mainboard , iModIdx		:= 0);
	MDP_Read												: 	FB_MDP_Read;
	SplitErrorId											:	FB_MDP_SplitErrorID;
	DstBuf													:	ARRAY[0..21] OF BYTE;
END_VAR

(* Read Mainboard Information 				V1.0	*)
(****************************************************)

(* Start Read *******************************************************)
	IF Execute
		AND state = 0
	THEN
		MB_Type												:= '';
		SerielNo											:= '';
		ProdDate											:= '';
		BootCount											:= 0;
		OpTime												:= 0;
		MinBoardTemp										:= 0;
		MaxBoardTemp										:= 0;
		MinInputVolt										:= 0;
		MaxInputVolt										:= 0;
		MB_Temp												:= 0;
		MEMSET(ADR(VoltLocation),0,SIZEOF(VoltLocation));
		MEMSET(ADR(VoltageValue),0,SIZEOF(VoltageValue));
		MEMSET(ADR(VoltageNominal),0,SIZEOF(VoltageNominal));
		VoltCount											:= 0;

		Busy												:= TRUE;
		Done												:= FALSE;
		Error												:= FALSE;
		ErrorId												:= 0;
		ErrorGrp											:= eMDP_Err_NoError;
		MDP_Read(bExecute := FALSE);
		MDP_ScanModules(
			bExecute			:= FALSE,
			nModuleType			:= eMDP_ModT_Mainboard,
			iModIdx				:= 0,
			tTimeout			:= timeout,
			sAmsNetId			:= AmsNetId,
			bBusy				=> ,
			bError				=> ,
			nErrID				=> ,
			nDynModuleId		=> ,
			iModuleTypeCount	=> ,
			iModuleCount		=> );

		MDP_ScanModules(bExecute:= TRUE);	
		state												:= 1;
		
	ELSIF NOT Execute
		AND State = 99
	THEN
		state												:= 0;
		Busy												:= FALSE;
		Done												:= FALSE;
		Error												:= FALSE;
		ErrorId												:= 0;
		ErrorGrp											:= eMDP_Err_NoError;
	END_IF


	CASE state OF
	0:
		;

	1:
		MDP_ScanModules();
		IF NOT MDP_ScanModules.bBusy
		THEN
			IF MDP_ScanModules.bError
			THEN
				Busy										:= FALSE;
				Error										:= TRUE;
				SplitErrorId(
					nErrID		:= MDP_ScanModules.nErrID,
					eErrGroup	=> ErrorGrp ,
					nErrCode	=> ErrorId);
				state										:= 99;
				MDP_ScanModules(bExecute := FALSE);
			ELSE
				MDP_Read(bExecute := FALSE);
				MDP_Read.stMDP_DynAddr.nArea				:= 16#8;
				MDP_Read.stMDP_DynAddr.nModuleId			:= MDP_ScanModules.nDynModuleId;
				MDP_Read.stMDP_DynAddr.nTableId				:= 1;
				MDP_Read.stMDP_DynAddr.nSubIdx				:= 0;
				idx											:= 1;
				state										:= 2;
			END_IF                                  		

		END_IF

	2:
		MDP_Read( pDstBuf	:= ADR(DstBuf), cbDstBufLen := SIZEOF(DstBuf));
		IF NOT MDP_Read.bBusy
		THEN
			IF MDP_Read.bError AND MDP_Read.bExecute
			THEN
				Busy										:= FALSE;
				Error										:= TRUE;
				SplitErrorId(
					nErrID		:= MDP_Read.nErrID,
					eErrGroup	=> ErrorGrp ,
					nErrCode	=> ErrorId);
				state										:= 99;
				MDP_Read(bExecute := FALSE);
			ELSE
				MDP_Read(bExecute := FALSE);
				CASE MDP_Read.stMDP_DynAddr.nTableId OF
				1:
					CASE MDP_Read.stMDP_DynAddr.nSubIdx OF
					0:
						MDP_Read.stMDP_DynAddr.nSubIdx		:= 1;

					1:
						MEMCPY(ADR(MB_Type), ADR(DstBuf), MIN(MDP_Read.nCount, SIZEOF(MB_Type)) );
						MDP_Read.stMDP_DynAddr.nSubIdx		:= 2;

					2:
						MEMCPY(ADR(SerielNo), ADR(DstBuf), MIN(MDP_Read.nCount, SIZEOF(SerielNo)) );
						MDP_Read.stMDP_DynAddr.nSubIdx		:= 3;

					3:
						MEMCPY(ADR(ProdDate), ADR(DstBuf), MIN(MDP_Read.nCount, SIZEOF(ProdDate)) );
						MDP_Read.stMDP_DynAddr.nSubIdx		:= 4;

					4:
						MEMCPY(ADR(BootCount), ADR(DstBuf), SIZEOF(BootCount));
						MDP_Read.stMDP_DynAddr.nSubIdx		:= 5;

					5:
						MEMCPY(ADR(OpTime), ADR(DstBuf), SIZEOF(OpTime));
						MDP_Read.stMDP_DynAddr.nSubIdx		:= 6;

					6:
						MEMCPY(ADR(MinBoardTemp), ADR(DstBuf), SIZEOF(MinBoardTemp));
						MDP_Read.stMDP_DynAddr.nSubIdx		:= 7;

					7:
						MEMCPY(ADR(MaxBoardTemp), ADR(DstBuf), SIZEOF(MaxBoardTemp));
						MDP_Read.stMDP_DynAddr.nSubIdx		:= 8;

					8:
						MEMCPY(ADR(MinInputVolt), ADR(DstBuf), SIZEOF(MinInputVolt));
						MDP_Read.stMDP_DynAddr.nSubIdx		:= 9;

					9:
						MEMCPY(ADR(MaxInputVolt), ADR(DstBuf), SIZEOF(MaxInputVolt));
						MDP_Read.stMDP_DynAddr.nSubIdx		:= 10;

					10:
						MEMCPY(ADR(MB_Temp), ADR(DstBuf), SIZEOF(MB_Temp));
						MDP_Read.stMDP_DynAddr.nSubIdx		:= 0;
						MDP_Read.stMDP_DynAddr.nTableId		:= 4;
					END_CASE

				4:
					CASE MDP_Read.stMDP_DynAddr.nSubIdx OF
					0:
						MEMCPY(ADR(VoltCount), ADR(DstBuf), SIZEOF(VoltCount) );
						IF VoltCount > 0 THEN
							MDP_Read.stMDP_DynAddr.nSubIdx	:= 1;
						ELSE						
							state							:= 3;
						END_IF

					1..255:
						MEMCPY(ADR(VoltLocation[MDP_Read.stMDP_DynAddr.nSubIdx]), ADR(DstBuf), SIZEOF(VoltLocation[MIN_VOLTAGE]));
						MDP_Read.stMDP_DynAddr.nSubIdx	:= MDP_Read.stMDP_DynAddr.nSubIdx + 1;
						
						IF MDP_Read.stMDP_DynAddr.nSubIdx > VoltCount
						THEN
							MDP_Read.stMDP_DynAddr.nSubIdx	:= 1;
							MDP_Read.stMDP_DynAddr.nTableId	:= 5;
						END_IF
					END_CASE

				5:
					CASE MDP_Read.stMDP_DynAddr.nSubIdx OF
					1..255:
						MEMCPY(ADR(VoltageValue[MDP_Read.stMDP_DynAddr.nSubIdx]), ADR(DstBuf), SIZEOF(VoltageValue[MIN_VOLTAGE]));
						MDP_Read.stMDP_DynAddr.nSubIdx	:= MDP_Read.stMDP_DynAddr.nSubIdx + 1;
						
						IF MDP_Read.stMDP_DynAddr.nSubIdx > VoltCount
						THEN
							MDP_Read.stMDP_DynAddr.nSubIdx	:= 1;
							MDP_Read.stMDP_DynAddr.nTableId	:= 6;
						END_IF
					END_CASE

				6:
					CASE MDP_Read.stMDP_DynAddr.nSubIdx OF
					1..255:
						MEMCPY(ADR(VoltageNominal[MDP_Read.stMDP_DynAddr.nSubIdx]), ADR(DstBuf), SIZEOF(VoltageNominal[MIN_VOLTAGE]));
						MDP_Read.stMDP_DynAddr.nSubIdx	:= MDP_Read.stMDP_DynAddr.nSubIdx + 1;
						
						IF MDP_Read.stMDP_DynAddr.nSubIdx > VoltCount
						THEN
							state							:= 3;
						END_IF
					END_CASE
				END_CASE

				MDP_Read(
					stMDP_DynAddr	:= ,		(* address to request subindex Count of AdressList *)
					pDstBuf			:= ADR(DstBuf),
					cbDstBufLen		:= SIZEOF(DstBuf),
					bExecute		:= NOT MDP_Read.bBusy AND state = 2,
					tTimeout		:= Timeout,
					sAmsNetId		:= AmsNetId,
					bBusy			=> ,
					bError			=> ,
					nErrId			=> );
			END_IF
		END_IF

	3: //Start lesen der IPC Seriennummer 
		MDP_Read.stMDP_DynAddr.nArea						:= INT_TO_BYTE(eMDP_Area_DeviceArea);
		MDP_Read.stMDP_DynAddr.nModuleId					:= 16#9F;
		MDP_Read.stMDP_DynAddr.nTableId						:= 16#00;
		MDP_Read.stMDP_DynAddr.nSubIdx						:= 16#00;
		
		MDP_Read(
			stMDP_DynAddr	:= ,		(* address to request subindex Count of AdressList *)
			pDstBuf			:= ADR(IPC_SerielNo),
			cbDstBufLen		:= SIZEOF(IPC_SerielNo),
			bExecute		:= NOT MDP_Read.bBusy,
			tTimeout		:= Timeout,
			sAmsNetId		:= AmsNetId,
			bBusy			=> ,
			bError			=> ,
			nErrId			=> );	
			
		state												:= 4;	
	
	4:
		MDP_Read( pDstBuf	:= ADR(IPC_SerielNo), cbDstBufLen := SIZEOF(IPC_SerielNo));
		IF NOT MDP_Read.bBusy
		THEN
			IF MDP_Read.bError AND MDP_Read.bExecute
			THEN
				Busy										:= FALSE;
				Error										:= TRUE;
				SplitErrorId(
					nErrID		:= MDP_Read.nErrID,
					eErrGroup	=> ErrorGrp ,
					nErrCode	=> ErrorId);
				state										:= 99;	
			ELSE			                        		
				Busy										:= FALSE;
				Done										:= TRUE;
				state										:= 99;
			END_IF
			MDP_Read(bExecute := FALSE);
			
		END_IF

	99: ;

	ELSE
		;
	END_CASE


	(* reset state for next start *)
	IF NOT Execute
		AND state = 99
	THEN
		state												:= 0;
	END_IF

(****************************************************************************************************)

END_FUNCTION_BLOCK

// ---- POUs/IpcDiag/MDP/InfoModuls/MDP_ReadModulList.TcPOU
{attribute 'no_check'}
FUNCTION_BLOCK MDP_ReadModulList EXTENDS FbBase
VAR_INPUT
	AmsNetId												: 	T_AmsNetId := '';	//AmsNetId as text
	Timeout													:	TIME := DEFAULT_ADS_TIMEOUT;	//Ads timeout
END_VAR                     								
VAR_OUTPUT                  								
	ModulCount												:	USINT;	//number of modules
	ModulType												:	ARRAY[0..255] OF E_MDP_ModuleType; //Index = Modul ID
	ErrorGrp												:	E_MDP_ErrGroup := eMDP_Err_NoError;
END_VAR                     								
VAR                         								
	MDP_Read												: 	FB_MDP_Read		:= (stMDP_DynAddr := (nArea := INT_TO_BYTE(eMDP_Area_DeviceArea), nModuleId := 16#02, nTableId := 16#00, nFlag := 16#00, nSubIdx := 16#00));
	SplitErrorId											:	FB_MDP_SplitErrorID;
	dwData													:	ARRAY [1..2] OF WORD;
END_VAR

(* Read list ob available moduls			V1.0	*)
(****************************************************)

(* Start read ************************************************)
	IF Execute
		AND state = 0
	THEN
		IF FALSE
		THEN (* Modultypen Liste *)
			MDP_Read.stMDP_DynAddr.nModuleId				:= 16#01;
		ELSE (* Modul ID Liste *)               			
			MDP_Read.stMDP_DynAddr.nModuleId				:= 16#02;
		END_IF                                  			
		MDP_Read.stMDP_DynAddr.nSubIdx						:= 0;
		MEMSET(ADR(ModulType),0,SIZEOF(ModulType));
		ModulCount											:= 0;
		Busy												:= TRUE;
		Done												:= FALSE;
		Error												:= FALSE;
		ErrorId												:= 0;
		ErrorGrp											:= eMDP_Err_NoError;
		
		MDP_Read(
			stMDP_DynAddr	:= ,		(* address to request subindex Count of AdressList *)
			pDstBuf			:= ADR(dwData),
			cbDstBufLen		:= SIZEOF(dwData),
			bExecute		:= FALSE,
			tTimeout		:= Timeout,
			sAmsNetId		:= AmsNetId,
			bBusy			=> ,
			bError			=> ,
			nErrId			=> );

		MDP_Read(bExecute	:= TRUE);
		state												:= 1;
	ELSIF NOT Execute
		AND State = 99
	THEN
		state												:= 0;
		Busy												:= FALSE;
		Done												:= FALSE;
		Error												:= FALSE;
		ErrorId												:= 0;
		ErrorGrp											:= eMDP_Err_NoError;
	END_IF


	CASE state OF
	0:
		;
	1:
		MDP_Read(pDstBuf := ADR(dwData), cbDstBufLen := SIZEOF(dwData));
		IF NOT MDP_Read.bBusy
		THEN
			IF MDP_Read.bError AND MDP_Read.bExecute
			THEN
				Busy										:= FALSE;
				Error										:= TRUE;
				SplitErrorId(
					nErrID		:= MDP_Read.nErrID,
					eErrGroup	=> ErrorGrp ,
					nErrCode	=> ErrorId);
				state										:= 99;
				MDP_Read(bExecute := FALSE);
			ELSE
				IF ModulCount = 0
				THEN (* Init Modul count *)
					ModulCount								:= WORD_TO_USINT(dwData[1]);
				ELSIF MDP_Read.stMDP_DynAddr.nSubIdx > 0
				THEN (* copy emlement dat					a *)
					ModulType[MDP_Read.stMDP_DynAddr.nSubIdx - 1] :=  dwData[2];					
				END_IF
				MDP_Read(bExecute := FALSE);
				MDP_Read.stMDP_DynAddr.nSubIdx:= MDP_Read.stMDP_DynAddr.nSubIdx + 1;
				IF MDP_Read.stMDP_DynAddr.nSubIdx > ModulCount
					OR MDP_Read.stMDP_DynAddr.nSubIdx > 255
				THEN
					Busy									:= FALSE;
					Done									:= TRUE;
					state									:= 99;
				ELSE
					MDP_Read(bExecute := TRUE,	pDstBuf	:= ADR(dwData), cbDstBufLen := SIZEOF(dwData));
				END_IF
			END_IF

		END_IF

	99: ;

	ELSE
		;
	END_CASE

	(* reset state for next start *)
	IF NOT Execute
		AND state = 99
	THEN
		state												:= 0;
	END_IF

(****************************************************************************************************)

END_FUNCTION_BLOCK

// ---- POUs/IpcDiag/MDP/InfoModuls/MDP_UPS.TcPOU
{attribute 'no_check'}
FUNCTION_BLOCK MDP_UPS EXTENDS FbBase
VAR_OUTPUT CONSTANT
(* Battery Power Status *)
	PS_UNKNOWN												:	INT := 0;
	PS_ONLINE												:	INT := 1;
	PS_ONBATTERIES											:	INT := 2;
	                    									
(* Com Status *)        									
	CS_UNKNOWN												:	INT := 0;
	CS_OK													:	INT := 1;
	CS_ERROR												:	INT := 2;

(* Battery Power Status *)
	BS_UNKNOWN												:	INT := 0;
	BS_OK													:	INT := 1;
	BS_CHANGE_BATTERY										:	INT := 2;
	
END_VAR
VAR_INPUT
	AmsNetId												: 	T_AmsNetId := '';	//AmsNetId
	Timeout													:	TIME := DEFAULT_ADS_TIMEOUT;	//Ads timeout
END_VAR
VAR_OUTPUT
(* UPS Data *)              								
	Model													:	STRING(30);	//model name
	VendorName												:	STRING(30);	//vendor name
	PowerStatus												:	INT := PS_UNKNOWN;
	ComStatus												:	INT := CS_UNKNOWN;
	BatteryStatus											:	INT := BS_UNKNOWN;
	BatteryCapacity											:	USINT; 		//in %
	BatteryRuntime											:	UDINT; 		//in sec
	PersPowerFailCounter									:	BOOL;		//TRUE when persistent power fail counter is activated
	PowerFailCounter										:	UDINT;		//number of power fails
	FanError												:	BOOL;		//Fan has error
	NoBattery												:	BOOL;		//No battery connected
	ErrorGrp												:	E_MDP_ErrGroup := eMDP_Err_NoError;

END_VAR                     								
VAR                         								
	idx														:	INT := 1;
	MDP_ScanModules											:	FB_MDP_ScanModules := ( nModuleType 	:= eMDP_ModT_UPS , iModIdx		:= 0);
	MDP_Read												: 	FB_MDP_Read;
	SplitErrorId											:	FB_MDP_SplitErrorID;
	DstBuf													:	ARRAY[0..31] OF BYTE;
END_VAR

	(* Read UPS Information 							V1.0	*)
	(***************************************************)

(* Start Read *******************************************************)
	IF Execute
		AND state = 0
	THEN
		Model												:= '';
		VendorName											:= '';
		PowerStatus											:= PS_UNKNOWN;
		ComStatus											:=	CS_UNKNOWN;
		BatteryStatus										:=	BS_UNKNOWN;
		BatteryCapacity										:= 0;
		BatteryRuntime										:= 0;
		PowerFailCounter									:= 0;
		PersPowerFailCounter								:= FALSE;
		FanError											:= FALSE;
		NoBattery											:= FALSE;
		Busy												:= TRUE;
		Done												:= FALSE;
		Error												:= FALSE;
		ErrorId												:= 0;
		ErrorGrp											:= eMDP_Err_NoError;
		MDP_Read(bExecute := FALSE);
		MDP_ScanModules(
			bExecute		:= NOT MDP_ScanModules.bExecute,
			nModuleType		:= eMDP_ModT_UPS,
			iModIdx			:= 0,
			tTimeout		:= timeout,
			sAmsNetId		:= AmsNetId,
			bBusy			=> ,
			bError			=> ,
			nErrID			=> ,
			nDynModuleId	=> ,
			iModuleTypeCount=> ,
			iModuleCount	=> );
			
		MDP_ScanModules(bExecute := TRUE);
		
		state												:= 1;
	ELSIF NOT Execute
		AND State = 99
	THEN
		state												:= 0;
		Busy												:= FALSE;
		Done												:= FALSE;
		Error												:= FALSE;
		ErrorId												:= 0;
		ErrorGrp											:= eMDP_Err_NoError;
	END_IF


	CASE state OF
	0:
		;
	1:
		MDP_ScanModules();
		IF NOT MDP_ScanModules.bBusy
		THEN
			IF MDP_ScanModules.bError
			THEN
				Busy										:= FALSE;
				Error										:= TRUE;
				SplitErrorId(
					nErrID		:= MDP_ScanModules.nErrID,
					eErrGroup	=> ErrorGrp ,
					nErrCode	=> ErrorId);
				state										:= 99;
				MDP_ScanModules(bExecute := FALSE);
			ELSE
				MDP_Read(bExecute := FALSE);
				MDP_Read.stMDP_DynAddr.nArea				:= 16#8;
				MDP_Read.stMDP_DynAddr.nModuleId			:= MDP_ScanModules.nDynModuleId;
				MDP_Read.stMDP_DynAddr.nTableId				:= 1;
				MDP_Read.stMDP_DynAddr.nSubIdx				:= 0;
				state										:= 2;
			END_IF

		END_IF

	2:
		MDP_Read( pDstBuf	:= ADR(DstBuf), cbDstBufLen := SIZEOF(DstBuf));
		IF NOT MDP_Read.bBusy
		THEN
			IF MDP_Read.bError AND MDP_Read.bExecute
			THEN
				Busy										:= FALSE;
				Error										:= TRUE;
				SplitErrorId(
					nErrID		:= MDP_Read.nErrID,
					eErrGroup	=> ErrorGrp ,
					nErrCode	=> ErrorId);
				state										:= 99;
				MDP_Read(bExecute := FALSE);
			ELSE
				MDP_Read(bExecute := FALSE);
				CASE MDP_Read.stMDP_DynAddr.nSubIdx	OF
				0:
					MDP_Read.stMDP_DynAddr.nSubIdx			:= 1;

				1:
					MEMCPY(ADR(Model), ADR(DstBuf), SIZEOF(Model) - 1);
					MDP_Read.stMDP_DynAddr.nSubIdx			:= 2;

				2:
					MEMCPY(ADR(VendorName), ADR(DstBuf), SIZEOF(VendorName) - 1);
					MDP_Read.stMDP_DynAddr.nSubIdx			:= 7;

				7:
					MEMCPY(ADR(PowerStatus), ADR(DstBuf), 1);
					MDP_Read.stMDP_DynAddr.nSubIdx			:= 8;

				8:
					MEMCPY(ADR(ComStatus), ADR(DstBuf), 1);
					MDP_Read.stMDP_DynAddr.nSubIdx			:= 9;

				9:
					MEMCPY(ADR(BatteryStatus), ADR(DstBuf), 1);
					MDP_Read.stMDP_DynAddr.nSubIdx			:= 10;

				10:
					MEMCPY(ADR(BatteryCapacity), ADR(DstBuf), SIZEOF(BatteryCapacity));
					MDP_Read.stMDP_DynAddr.nSubIdx			:= 11;

				11:
					MEMCPY(ADR(BatteryRuntime), ADR(DstBuf), SIZEOF(BatteryRuntime));
					MDP_Read.stMDP_DynAddr.nSubIdx			:= 12;

				12:
					MEMCPY(ADR(PersPowerFailCounter), ADR(DstBuf), SIZEOF(PersPowerFailCounter));
					MDP_Read.stMDP_DynAddr.nSubIdx			:= 13;

				13:
					MEMCPY(ADR(PowerFailCounter), ADR(DstBuf), SIZEOF(PowerFailCounter));
					MDP_Read.stMDP_DynAddr.nSubIdx			:= 14;

				14:
					MEMCPY(ADR(FanError), ADR(DstBuf), SIZEOF(FanError));
					MDP_Read.stMDP_DynAddr.nSubIdx			:= 15;

				15:
					MEMCPY(ADR(NoBattery), ADR(DstBuf), SIZEOF(NoBattery));
					Busy									:= FALSE;
					Done									:= TRUE;
					state									:= 99;
                                                        	
				ELSE                                    	
					Busy									:= FALSE;
					Done									:= TRUE;
					state									:= 99;
				END_CASE

				MDP_Read(
					stMDP_DynAddr	:= ,(* address to request subindex Count of AdressList *)
					pDstBuf			:= ADR(DstBuf),
					cbDstBufLen		:= SIZEOF(DstBuf),
					bExecute		:= NOT MDP_Read.bBusy AND state = 2,
					tTimeout		:= Timeout,
					sAmsNetId		:= AmsNetId,
					bBusy			=> ,
					bError			=> ,
					nErrId			=> );
			END_IF
		END_IF

	99: ;

	ELSE
		;
	END_CASE

	(* reset state for next start *)
	IF NOT Execute
		AND state = 99
	THEN
		state												:= 0;
	END_IF

(****************************************************************************************************)

END_FUNCTION_BLOCK

// ---- POUs/IpcDiag/MDP/MDP_IpcDiag.TcPOU
{attribute 'no_check'}
//General IPC diagnosis based on Beckhoff MDP - invalid values are reported via EventLogger 
//based on Tc2_MDP.lib - please see Beckhoff documentation for further information about Tc2_MDP.lib (IPC diagnostics)
//EventHandlingGrp10 instance used inside
//Info:
// 0x   	a    	nn   	x   
// 0x   	8   	03   	1   
// a 	= Area Code (e.g. 8 = Configuration Area) 
// nn 	= Modul-ID (e.g. dynamic modul id from list F020) 
// x	= Tabel id (e.g. 1 = Table 0x8nn1 - NIC Properties at area code 8) 
FUNCTION_BLOCK MDP_IpcDiag
VAR CONSTANT
	MIN_CPU													:	INT := 1;
	MAX_CPU													:	INT := 4;
	                    									
	MIN_FAN													:	INT := 1;
	MAX_FAN													:	INT := 4;
	                    									
	MIN_VOLTAGE												:	INT := 1;
	MAX_VOLTAGE												:	INT := 8;		
END_VAR                 									
VAR_INPUT               									
	Enable													:	BOOL := FALSE;	//FB will be processed as long as enable is TRUE 
	CycleTime												:	TIME := T#100MS; //Delay between ads call to read a single value 
	AmsNetId												: 	T_AmsNetId := ''; //Ams net Id
	Timeout													: 	TIME := DEFAULT_ADS_TIMEOUT; //Ads timeout
{attribute 'displaymode':='bin'}
	FanMask													:	BYTE := 2#0000_0011; //Installed fans inside the PC 
	
//Threshold values 	    									
	MinSpeedFan												:	INT := 2500; 	//rpm
	MaxTempMB												:	INT := 85; 		//°C
	MaxTempCPU												:	INT := 100; 	//°C
	TempWarningThreshold									:	INT := 10; 		//°C
	VoltageFactor											:	LREAL := 0.7; 	//% of nominal voltage before an error occurs
END_VAR                 									
VAR_OUTPUT              										                									
	MB_Temp													:	INT; //Motherboard temp with one decimal digit  
	Voltage_Count											:	INT := 0; //count of voltage measurement points with one decimal digit 
	MB_NominalVoltage										:	ARRAY[MIN_VOLTAGE..MAX_VOLTAGE] OF INT; //in mV
	MB_Voltage												:	ARRAY[MIN_VOLTAGE..MAX_VOLTAGE] OF INT;  //in mV
	CPU_Count												:	INT := 0; //Readed number of CPUs
	CPU_Temp												:	ARRAY[MIN_CPU..MAX_CPU] OF INT; //cpu temperatur with one decimal digit
	FAN_Count												:	INT := 0; //Number of FANs in config. Note, the number may be two where only the second fan is p
	FAN_Speed												:	ARRAY[MIN_FAN..MAX_FAN] OF INT; //in rpm for each available fan
	OsImage													:	STRING; //Image version 
	ExecutionTime											:	TIME; 	//Cylce time to execute function block        
	Busy													:	BOOL;	//Busy is TRUE at the rising edge of Enable and stays TRUE as long as the FB is performing any action. 
	Valid													:	BOOL;	//data valid
	Error													:	BOOL;	//Rising edge of Error informs that an error occurred during the execution of the Function Block 
{attribute 'displaymode':='hex'}
	ErrorId													:	UDINT;	//Error identification - see documentation about IPC diagnostic for further detailed informantion 
	ErrorGrp												:	E_MDP_ErrGroup := eMDP_Err_NoError; //MDP Error code - see Beckhoff documentation MDP for further informantion
END_VAR	
VAR
(* cache variables ************************************************************)
	state													:	INT := 0;
	
	dwData													:	ARRAY [1..2] OF WORD;
	                    									
	MemLen													:	BYTE := 0;
	MemModIdMB												:	BYTE;
	MemModIdCPU												:	ARRAY[MIN_CPU..MAX_CPU] OF BYTE;
	MemModIdFan												:	ARRAY[MIN_FAN..MAX_FAN] OF BYTE;
	MEmModIdUPS												:	BYTE;
	MemMBSubIdxVoltage										:	ARRAY[MIN_VOLTAGE..MAX_VOLTAGE] OF BYTE;
	MemTimeStartCycle										:	TIME;
	MemErrState												:	INT := 0;
	
(* timer ***************************************************************************)
	TON_Cycle												:	TON;
	
(* function-blocks *****************************************************************)
	MDP_Read												: 	FB_MDP_Read		:= (tTimeout := DEFAULT_ADS_TIMEOUT, stMDP_DynAddr := (nArea := INT_TO_BYTE(eMDP_Area_DeviceArea), nModuleId := 16#02, nTableId := 16#00, nFlag := 16#00, nSubIdx := 16#00));
	SplitErrorId											:	FB_MDP_SplitErrorID;
	
(* internal used variables **********************************************************)
	i,k														:	INT;

END_VAR

(* MDP IPC diag compact						V1.1	*)
(****************************************************)

(* Sequence *******************************************************)
IF Enable
THEN
	CASE state OF
	0:	
		IF NOT MDP_Read.bBusy
			AND NOT Error
		THEN
			Busy											:= TRUE;
			Valid											:= FALSE;
		
			Fan_Count										:= 0;
			CPU_Count										:= 0;
			Voltage_Count									:= 0;
			MemLen											:= 0;
			MB_Temp											:= 0;
			MEMSET(ADR(MB_Voltage),0,SIZEOF(MB_Voltage));
			MEMSET(ADR(CPU_Temp),0,SIZEOF(CPU_Temp));
			MEMSET(ADR(FAN_Speed),0,SIZEOF(FAN_Speed));
			MEMSET(ADR(MemModIdCPU),0,SIZEOF(MemModIdCPU));
			MEMSET(ADR(MemModIdFan),0,SIZEOF(MemModIdFan));
			MEMSET(ADR(MemMBSubIdxVoltage),0,SIZEOF(MemMBSubIdxVoltage));
			MEMSET(ADR(MB_NominalVoltage),0,SIZEOF(MB_NominalVoltage));
			
			MDP_Read.stMDP_DynAddr.nArea					:= INT_TO_BYTE(eMDP_Area_GeneralArea);
			MDP_Read.stMDP_DynAddr.nModuleId				:= 16#00;
			MDP_Read.stMDP_DynAddr.nTableId					:= 16#0A;
			MDP_Read.stMDP_DynAddr.nSubIdx					:= 16#00;
                                                    			                                        		
			state											:= 1;
		ELSE
			MDP_Read(bExecute := FALSE);	
		END_IF
		
	1:
	//Read OS version 	
		MDP_Read(bExecute := TRUE , pDstBuf := ADR(OsImage), cbDstBufLen := SIZEOF(OsImage));
		IF NOT MDP_Read.bBusy
		THEN
			IF MDP_Read.bError AND MDP_Read.bExecute
			THEN
				Busy										:= FALSE;
				Error										:= TRUE;
				SplitErrorId(
					nErrID		:= MDP_Read.nErrID,
					eErrGroup	=> ErrorGrp ,
					nErrCode	=> ErrorId);
				MemErrState									:= state;		
				state										:= 99;
				MDP_Read(bExecute := FALSE);
			ELSE //Os Image readed
				k											:= UDINT_TO_INT(MDP_Read.nCount + 1);	
				OsImage[k]									:= 0; //Terminate string
				MDP_Read(bExecute := FALSE);	
				
				//Deveice area F + Modul Id 02 + Tabel Id = 0 -> Index 0xF020 – Modul ID Liste in deveice area
				MDP_Read.stMDP_DynAddr.nArea				:= INT_TO_BYTE(eMDP_Area_DeviceArea); //Index F
				MDP_Read.stMDP_DynAddr.nModuleId			:= 16#02; //Modul id 02 in Config area dynamic modul ids are used!
				MDP_Read.stMDP_DynAddr.nTableId				:= 16#00; //Table Id 0
				MDP_Read.stMDP_DynAddr.nSubIdx				:= 16#00; //Len = number of dyn moduls			
				state										:= 2;								
			END_IF
		END_IF		
		
	2: // search list with dynamic moduls
		MDP_Read(bExecute := TRUE, pDstBuf := ADR(dwData), cbDstBufLen := SIZEOF(dwData));
		IF NOT MDP_Read.bBusy
		THEN
			IF MDP_Read.bError AND MDP_Read.bExecute
			THEN
				Busy										:= FALSE;
				Error										:= TRUE;
				SplitErrorId(
					nErrID		:= MDP_Read.nErrID,
					eErrGroup	=> ErrorGrp ,
					nErrCode	=> ErrorId);
				MemErrState									:= state;	
				state										:= 99;
				MDP_Read(bExecute := FALSE);
			ELSE
				IF MemLen = 0
				THEN (* Init Modul count *)
					MemLen									:= WORD_TO_BYTE(dwData[1]);
				ELSIF MDP_Read.stMDP_DynAddr.nSubIdx > 0
				THEN (* copy emlement dat					a *)
					CASE dwData[2] OF //High word = Modul type, Low word = Modul Id
					Tc2_MDP.E_MDP_ModuleType.eMDP_ModT_Mainboard:
						MemModIdMB		 					:= WORD_TO_BYTE(dwData[1]);		

					Tc2_MDP.E_MDP_ModuleType.eMDP_ModT_UPS:
						MEmModIdUPS							:= WORD_TO_BYTE(dwData[1]);

					Tc2_MDP.E_MDP_ModuleType.eMDP_ModT_CPU:
						CPU_Count							:= CPU_Count + 1;
						MemModIdCPU[CPU_Count]				:= WORD_TO_BYTE(dwData[1]);

					Tc2_MDP.E_MDP_ModuleType.eMDP_ModT_Fan:
						Fan_Count							:= Fan_Count + 1;
						MemModIdFan[Fan_Count]				:= WORD_TO_BYTE(dwData[1]);
												
					ELSE
						; 
					END_CASE				
				END_IF
				MDP_Read(bExecute := FALSE);
				MDP_Read.stMDP_DynAddr.nSubIdx:= MDP_Read.stMDP_DynAddr.nSubIdx + 1;
				IF MDP_Read.stMDP_DynAddr.nSubIdx > MemLen
					OR MDP_Read.stMDP_DynAddr.nSubIdx > 255
				THEN
					state									:= SEL(MemModIdMB > 0 , 9 , 3);								
				ELSE
					MDP_Read(bExecute := TRUE,	pDstBuf	:= ADR(dwData), cbDstBufLen := SIZEOF(dwData));
				END_IF
			END_IF

		END_IF
				
	3: //reading motherboardconfig (SubIndex Voltage)
		MDP_Read.stMDP_DynAddr.nArea						:= INT_TO_BYTE(eMDP_Area_ConfigArea);
		MDP_Read.stMDP_DynAddr.nModuleId					:= INT_TO_BYTE(MemModIdMB);
		MDP_Read.stMDP_DynAddr.nTableId						:= 16#04;
		MDP_Read.stMDP_DynAddr.nSubIdx						:= 16#00;
		MemLen												:= 0;
		i													:= 0;
		
		MDP_Read(
			stMDP_DynAddr	:= ,		(* address to request subindex Count of AdressList *)
			pDstBuf			:= ADR(dwData[1]),
			cbDstBufLen		:= SIZEOF(dwData[1]),
			bExecute		:= NOT MDP_Read.bBusy,
			tTimeout		:= ,
			sAmsNetId		:= AmsNetId,
			bBusy			=> ,
			bError			=> ,
			nErrId			=> );	
			
		state												:= 4;	
	
	4: 
		MDP_Read(pDstBuf := ADR(dwData[1]), cbDstBufLen := SIZEOF(dwData[1]));
		IF NOT MDP_Read.bBusy
		THEN
			IF MDP_Read.bError AND MDP_Read.bExecute
			THEN
				Busy										:= FALSE;
				Error										:= TRUE;
				SplitErrorId(
					nErrID		:= MDP_Read.nErrID,
					eErrGroup	=> ErrorGrp ,
					nErrCode	=> ErrorId);
				MemErrState									:= state;		
				state										:= 99;
				MDP_Read(bExecute := FALSE);
			ELSE
				IF MemLen = 0
				THEN (* Init Entry count *)
					MemLen									:= WORD_TO_BYTE(dwData[1]);
				ELSE 
					MDP_Read(bExecute := FALSE);
					(* copy emlement data
						00 = LOCATION_UNKNOWN
						01 = LOCATION_OTHER
						02 = LOCATION_PROCESSOR
						03 = LOCATION_DISK
						04 = LOCATION_SYSTEM_MANAGEMENT_MODULE
						05 = LOCATION_MOTHERBOARD
						06 = LOCATION_MEMORY_MODULE
						07 = LOCATION_POWER_SUPPLY
						08 = LOCATION_ADDIN_CARD
						09 = LOCATION_FRONT_PANEL_BOARD
						10 = LOCATION_BACK_PANEL_BOARD
						11 = LOCATION_PERIPHERIE
						12 = LOCATION_CHASSIS
						13 = LOCATION_BATTERY
						14 = LOCATION_UPS
						15 = LOCATION_GRAFFIC_BOARD
						16 = LOCATION_SUPERIO
						17 = LOCATION_CHIPSET
					*)

				
					CASE dwData[1] OF
					7, //PowerSupply			
					13: //Battery
						Voltage_Count						:= Voltage_Count + 1;
						MemMBSubIdxVoltage[Voltage_Count]	:= MDP_Read.stMDP_DynAddr.nSubIdx; 
					ELSE
						; 
					END_CASE			
					MDP_Read.stMDP_DynAddr.nSubIdx			:= MDP_Read.stMDP_DynAddr.nSubIdx + 1; 				
							
					IF MDP_Read.stMDP_DynAddr.nSubIdx > MemLen
						OR MDP_Read.stMDP_DynAddr.nSubIdx > 255
						OR Voltage_Count >= MAX_Voltage
					THEN
						IF Voltage_Count > 0
						THEN
							i 								:= MIN_VOLTAGE;
							MDP_Read.stMDP_DynAddr.nTableId	:= 16#06;
							MDP_Read.stMDP_DynAddr.nSubIdx	:= MemMBSubIdxVoltage[i];
							MDP_Read(bExecute := TRUE,	pDstBuf	:= ADR(dwData[1]), cbDstBufLen := SIZEOF(dwData[1]));												
							state							:= 5;				
						ELSE
							state							:= 9;	
						END_IF
				
					ELSE
						MDP_Read(bExecute := TRUE,	pDstBuf	:= ADR(dwData[1]), cbDstBufLen := SIZEOF(dwData[1]));
					END_IF
				END_IF
			END_IF

		END_IF	

	5:	//Nominal Voltage lesen
		MDP_Read(pDstBuf := ADR(dwData[1]), cbDstBufLen := SIZEOF(dwData[1]));
		IF NOT MDP_Read.bBusy
		THEN
			IF MDP_Read.bError AND MDP_Read.bExecute
			THEN
				Busy										:= FALSE;
				Error										:= TRUE;
				SplitErrorId(
					nErrID		:= MDP_Read.nErrID,
					eErrGroup	=> ErrorGrp ,
					nErrCode	=> ErrorId);
				MemErrState									:= state;		
				state										:= 99;
				MDP_Read(bExecute := FALSE);
			ELSE //Nominal Volage
				MDP_Read(bExecute := FALSE);
				MB_NominalVoltage[i]						:= WORD_TO_INT(dwData[1]); 
				i 											:= i + 1;
				IF i > MAX_VOLTAGE
					OR i > Voltage_Count
				THEN //Ende der Bearbeitung
					state									:= 9;								
				ELSE
					MDP_Read.stMDP_DynAddr.nSubIdx			:= MemMBSubIdxVoltage[i];
					MDP_Read(bExecute := TRUE,	pDstBuf	:= ADR(dwData[1]), cbDstBufLen := SIZEOF(dwData[1]));
				END_IF
			END_IF

		END_IF	
							
	//Start Cylce Read
	9: 	
		TON_Cycle(IN := FALSE);
		MemTimeStartCycle									:= T#0MS;
		i													:= 0;
		state												:= 10;	
		
	//Start lesen der Zyklischen Daten 
	10..90: 
		MDP_Read(pDstBuf := ADR(dwData[1]), cbDstBufLen := SIZEOF(dwData[1]));
		IF NOT MDP_Read.bBusy
		THEN			
			IF MDP_Read.bError AND MDP_Read.bExecute
			THEN
				Busy										:= FALSE;
				Error										:= TRUE;
				SplitErrorId(
					nErrID		:= MDP_Read.nErrID,
					eErrGroup	=> ErrorGrp ,
					nErrCode	=> ErrorId);
				MemErrState									:= state;	
				state										:= 99;
				MDP_Read(bExecute := FALSE);
			ELSIF NOT TON_Cycle.IN
			THEN		
				MDP_Read(bExecute := FALSE);
				CASE state OF
				10:
					MDP_Read.stMDP_DynAddr.nModuleId		:= MemModIdMB;
					MDP_Read.stMDP_DynAddr.nTableId			:= 16#01;
					MDP_Read.stMDP_DynAddr.nSubIdx			:= 10;
					dwData[1]								:= 0;	
					TON_Cycle.IN							:= MDP_Read.stMDP_DynAddr.nModuleId > 0;			
					state									:= 11;
								
				11: 
					MB_Temp									:= WORD_TO_INT(dwData[1]); //Daten sichern
					
					i 										:= MIN_VOLTAGE;	
					IF Voltage_Count > 0
					THEN					
						MDP_Read.stMDP_DynAddr.nModuleId	:= MemModIdMB;
						MDP_Read.stMDP_DynAddr.nTableId		:= 16#05;
						MDP_Read.stMDP_DynAddr.nSubIdx		:= MemMBSubIdxVoltage[i];
						TON_Cycle.IN						:= MDP_Read.stMDP_DynAddr.nModuleId > 0;	
					ELSE
						dwData[1]							:= 0;	
					END_IF						
					
					state									:= 12;		
			
				12:
					MB_Voltage[i]							:= WORD_TO_INT(dwData[1]); //Daten sichern
				
					i 										:= i + 1;	
					IF i > Voltage_Count
					THEN //CPUTemp lesen 
						i									:= MIN_CPU;
						MDP_Read.stMDP_DynAddr.nModuleId	:= MemModIdCPU[i];
						MDP_Read.stMDP_DynAddr.nTableId		:= 16#01;
						MDP_Read.stMDP_DynAddr.nSubIdx		:= 3;
						TON_Cycle.IN						:= MDP_Read.stMDP_DynAddr.nModuleId > 0;		
						state								:= 13;					
					ELSE //weiter Voltage lesen
						MDP_Read.stMDP_DynAddr.nModuleId	:= MemModIdMB;
						MDP_Read.stMDP_DynAddr.nTableId		:= 16#05;
						MDP_Read.stMDP_DynAddr.nSubIdx		:= MemMBSubIdxVoltage[i];	
						TON_Cycle.IN						:= MDP_Read.stMDP_DynAddr.nModuleId > 0;		
					END_IF								
			
				13: 
					CPU_Temp[i]								:= WORD_TO_INT(dwData[1]);
					
					i 										:= i + 1;	
					IF i > CPU_Count //Start next read
					THEN //Fan auslesen 	
						IF Fan_Count > 0
						THEN
							i								:= MIN_FAN;
							
							MDP_Read.stMDP_DynAddr.nModuleId:= MemModIdFan[i];
							MDP_Read.stMDP_DynAddr.nTableId	:= 16#01;
							MDP_Read.stMDP_DynAddr.nSubIdx	:= 1;		
							TON_Cycle.IN					:= MDP_Read.stMDP_DynAddr.nModuleId > 0;			
						ELSE
							dwData[1]						:= 0;				
						END_IF
						
						state								:= 14;
						
					ELSE //CPU weiter auslesen
						MDP_Read.stMDP_DynAddr.nModuleId	:= MemModIdCPU[i];
						MDP_Read.stMDP_DynAddr.nTableId		:= 16#01;
						MDP_Read.stMDP_DynAddr.nSubIdx		:= 3;		
						TON_Cycle.IN						:= MDP_Read.stMDP_DynAddr.nModuleId > 0;						
					END_IF			
				
				14: 
					FAN_Speed[i]							:= WORD_TO_INT(dwData[1]);
					
					i 										:= i + 1;	
					IF i > Fan_Count
					THEN //CPU Usage auslesen
						(*
						i									:= MIN_CPU;
						MDP_Read.stMDP_DynAddr.nModuleId	:= MemModIdCPU[i];
						MDP_Read.stMDP_DynAddr.nTableId		:= 16#01;
						MDP_Read.stMDP_DynAddr.nSubIdx		:= 2;
						*)
						TON_Cycle.IN						:= MDP_Read.stMDP_DynAddr.nModuleId > 0;		
					//	state								:= 15;
						state								:= 90;	//final state in this section		
					
					ELSE //Fan weiter auslesen
						MDP_Read.stMDP_DynAddr.nModuleId	:= MemModIdFan[i];
						MDP_Read.stMDP_DynAddr.nTableId		:= 16#01;
						MDP_Read.stMDP_DynAddr.nSubIdx		:= 1;
						TON_Cycle.IN						:= MDP_Read.stMDP_DynAddr.nModuleId > 0;						
					END_IF				
				
				(*
				15:
					CPU_Usage[i]							:= WORD_TO_USINT(dwData[1]);
					
					i 										:= i + 1;	
					IF i > CPUCount
					THEN //Ups status auslesen 	
						IF MEmModIdUPS <> 0
						THEN
							MDP_Read.stMDP_DynAddr.nModuleId:= MEmModIdUPS;
							MDP_Read.stMDP_DynAddr.nTableId	:= 16#01;
							MDP_Read.stMDP_DynAddr.nSubIdx	:= 7;	
							TON_Cycle.IN					:= MDP_Read.stMDP_DynAddr.nModuleId > 0;
						ELSE
							dwData[1]						:= 0;								
						END_IF					
						state								:= 16;	
						
					ELSE //CPU weiter auslesen
						MDP_Read.stMDP_DynAddr.nModuleId	:= MemModIdCPU[i];
						MDP_Read.stMDP_DynAddr.nTableId		:= 16#01;
						MDP_Read.stMDP_DynAddr.nSubIdx		:= 2;		
						TON_Cycle.IN						:= MDP_Read.stMDP_DynAddr.nModuleId > 0;						
					END_IF	
			
				16:
					UPS_PowerStatus							:= WORD_TO_INT(dwData[1]);
					state									:= state * -1;	
				*)
				ELSE //90			
					Valid									:= TRUE;
					ExecutionTime	 						:= TIME() - MemTimeStartCycle;
					MemTimeStartCycle 						:= T#0MS;
					state									:= 10;	
				END_CASE
			END_IF
			TON_Cycle(PT := CycleTime);
			MDP_Read(bExecute := TON_Cycle.Q,	pDstBuf	:= ADR(dwData), cbDstBufLen := SIZEOF(dwData));
			
			IF MDP_Read.bExecute 
			THEN 
				TON_Cycle(IN := FALSE); 		
			END_IF 
			
			IF MemTimeStartCycle = T#0MS
			THEN
				MemTimeStartCycle 							:= TIME();	
			END_IF
			
		END_IF
			
	//Error State	
	99:	
		; //Wait for disable
				
	ELSE
		;
	END_CASE
ELSE //Not Enable
	state													:= 0;
	Error													:= FALSE;
	ErrorId													:= 0;
	ErrorGrp												:= eMDP_Err_NoError;
	Busy													:= FALSE;
	Valid													:= FALSE;
	MDP_Read(bExecute := FALSE);

END_IF			

(****************************************************************************************************)

END_FUNCTION_BLOCK

// ---- POUs/IpcDiag/UPSStatus.TcPOU
{attribute 'no_check'}
//General UPS function block to make use of differenty types of utility power supplies 
//Requiered libs : Tc2_SUPS, Tc2_IoFunctions
FUNCTION_BLOCK UPSStatus
VAR_OUTPUT CONSTANT
	MODE_SUPS_CB3011										:	INT := 0; //SUPS for CB3011 Motherboard
	MODE_SUPS_CX50X0										:	INT := 1; //SUPS for CX50X0
	MODE_SUPS_CX51X0										:	INT := 2; //SUPS for CX51X0
	MODE_SUPS_CX9020										:	INT := 3; //SUPS for CX9020
	MODE_SUPS_BAPI											:	INT := 4; //SUPS for BAPI
	MODE_UPS_BA												:	INT := 5; //BA UPS Controller CP903x-Card (PCI/ISA) | Beckhoff P24Vxxxx USV | With Beckhoff Industrial PC's delivered APC UPS models supporting smart protocol and configured with Windows UPS Service
	MODE_UPS_EXTERN_OK										:	INT := 6; //External UPS controller connected via one Digital Input -> TRUE=PowerOK
	MODE_UPS_EXTERN_FAIL									:	INT := 7; //External UPS controller connected via one Digital Input -> TRUE=PowerFAIL
END_VAR                     								
VAR_INPUT                   													
	Enable													: 	BOOL := FALSE;		// FB will be processed as long as enable is TRUE 
	NetId													: 	T_AmsNetId 	:= '';	// AmsNet id
	Port													: 	T_AmsPort 	:= 851; // TC3 PLC RT1 = 851.... , 0 = Windows UPS service 
	Timeout													: 	TIME := DEFAULT_ADS_TIMEOUT; // Ads timeout / PowerOK/Fault delay at mode = MODE_UPS_EXTERN
	Mode													: 	INT(MODE_SUPS_CB3011..MODE_UPS_EXTERN_FAIL) := MODE_UPS_BA; // Select used UPS type
	UpsMode													: 	E_S_UPS_Mode := eSUPS_WrPersistData_Shutdown; // Used by FB_S_UPS instances and adaped for modes <> MODE_SUPS  
END_VAR
VAR_OUTPUT
	BatteryReplace											:	BOOL;
	PowerFailDetect											:	BOOL; 	//TRUE when power fail is detected 
	Status													:	E_S_UPS_State := eSUPS_PowerOK; //Reports the status of utility-supplied power into the UPS. 
	Error													:	BOOL;		//Rising edge of Error informs that an error occurred during the execution of the Function Block  	
{attribute 'displaymode':='hex'}
	ErrorID													:	UDINT; 	//Error identification 
END_VAR      
VAR              
//local *****************************************************************
	State													: 	INT := 0;
	DigInput										AT %I*	: 	BOOL; //Hardware signal for OK/NOK depending on selected UpsMode
	
//Trigger ***************************************************************

//Timer ****************************************************************
	TonPowerOff												: 	TON;	
//Instances **********************************************************  
	UPSPowerStatus											: 	FB_GetUpsStatus;
	SUPSPowerStatus_CB3011									: 	FB_S_UPS_CB3011 		:= (ePersistentMode := SPDM_2PASS);
	SUPSPowerStatus_CX50X0									: 	FB_S_UPS 				:= (iUPSPort := 16#4A8 ,ePersistentMode := SPDM_2PASS);	
	SUPSPowerStatus_CX51x0									: 	FB_S_UPS_CX51x0 		:= (iUPSPort := 16#588 ,ePersistentMode := SPDM_2PASS);
	SUPSPowerStatus_CX9020									: 	FB_S_UPS_CX9020_U900 	:= (ePersistentMode := SPDM_2PASS);
	SUPSPowerStatus_BAPI									: 	FB_S_UPS_BAPI			:= (ePersistentMode := SPDM_2PASS);
	ShutDown												: 	NT_Shutdown;
	WritePersistentData										: 	FB_WritePersistentData := (Mode := SPDM_2PASS);	
	TcStop													: 	TC_Stop;
//Dummy *****************************************************************)       								

END_VAR

	(* UPS Wrapper										*)
	(****************************************************)

(* Sequence *************************************************************************)
IF Enable THEN
	CASE state OF	
	0:
		CASE MODE OF
		MODE_SUPS_CB3011:
			SUPSPowerStatus_CB3011(
				sNetID				:= NetId,
				iPLCPort			:= Port,
				tTimeout			:= ,
				eUpsMode			:= UpsMode,
				ePersistentMode		:= ,
				tRecoverTime		:= ,
				bPowerFailDetect	=> PowerFailDetect,
				eState				=> Status);		
		
		MODE_SUPS_CX50X0:
			SUPSPowerStatus_CX50X0(
				sNetID				:= NetId,
				iPLCPort			:= Port,
				iUPSPort			:= ,
				tTimeout			:= ,
				eUpsMode			:= UpsMode,
				ePersistentMode		:= ,
				tRecoverTime		:= ,
				bPowerFailDetect	=> PowerFailDetect,
				eState				=> Status);		
			
		MODE_SUPS_CX51X0:
			SUPSPowerStatus_CX51x0(
				sNetID				:= NetId,
				iPLCPort			:= Port,
				iUPSPort			:= ,
				tTimeout			:= ,
				eUpsMode			:= UpsMode,
				ePersistentMode		:= ,
				tRecoverTime		:= ,
				bPowerFailDetect	=> PowerFailDetect,
				eState				=> Status);		
			
		MODE_SUPS_CX9020:
			SUPSPowerStatus_CX9020(
				sNetID				:= NetId,
				iPLCPort			:= Port,
				tTimeout			:= ,
				eUpsMode			:= UpsMode,
				ePersistentMode		:= ,
				tRecoverTime		:= ,
				bPowerFailDetect	=> PowerFailDetect,
				eState				=> Status);		
				
		MODE_SUPS_BAPI:
			SUPSPowerStatus_BAPI(
				sNetID				:= NetId,
				iPLCPort			:= Port,
				tTimeout			:= ,
				eUpsMode			:= UpsMode,
				ePersistentMode		:= ,
				tRecoverTime		:= ,
				bPowerFailDetect	=> PowerFailDetect,
				eState				=> Status);				

		MODE_UPS_EXTERN_OK,
		MODE_UPS_EXTERN_FAIL:
			TonPowerOff(
				IN					:= SEL(MODE = MODE_UPS_EXTERN_OK, DigInput, NOT DigInput), 
				PT					:= Timeout, 
				Q 					=> PowerFailDetect);
			Status											:= SEL(TonPowerOff.IN, eSUPS_PowerOK, eSUPS_WaitForRecover);
			IF TonPowerOff.Q                                
			THEN				                            
				Status										:= eSUPS_PowerFailure;
				state										:= 900;
			END_IF 
			
		MODE_UPS_BA:		
			UPSPowerStatus(
				sNetId				:= NetId, 
				nPort				:= 0, 
				bEnable				:= TRUE, 
				bValid				=> , 
				bError				=> Error, 
				nErrId				=> ErrorID);
			BatteryReplace									:= UPSPowerStatus.stStatus.eBatteryStatus = E_BatteryStatus.BatteryReplace AND UPSPowerStatus.bValid;
			CASE UPSPowerStatus.stStatus.ePowerStatus OF 
			PowerUnknownStatus: 			// The status of power is unknown
				PowerFailDetect								:= FALSE;
				Status										:= eSUPS_PowerOK;	
 			PowerOnLine: 		 		  	// Power is OK
				PowerFailDetect								:= FALSE;
				Status										:= eSUPS_PowerOK;
   			PowerOnBattery:					// A power failure has occurred
				PowerFailDetect								:= UPSPowerStatus.bValid;
				Status										:= eSUPS_PowerFailure;
				state										:= 900;
			END_CASE
	
		ELSE
			state											:= 0;
			Error											:= TRUE;
			ErrorID											:= 1798;	
			PowerFailDetect									:= FALSE;		
			Status											:= eSUPS_PowerFailure;		
		END_CASE
		
	//Shutdown OS and stop TC ************************************************************)
	900: 
		ShutDown(START := FALSE); TcStop(Stop := FALSE); WritePersistentData(Start := FALSE);
		CASE UpsMode OF
		eSUPS_WrPersistData_NoShutdown:
			WritePersistentData(Start := TRUE, Port := Port);		
			status											:= eSUPS_WritePersistentData;
		eSUPS_ImmediateShutdown:
			ShutDown(START := TRUE, TMOUT := T#3S); 
			status											:= eSUPS_QuickShutdown;			
		ELSE //eSUPS_WrPersistData_Shutdown
			ShutDown(START := TRUE, TMOUT := T#3S);
			status											:= eSUPS_WritePersistentData;
		END_CASE
		state												:= state + 1;	
											
	901:// Wait for shutdown started     
		shutDown();  WritePersistentData();  																		
		IF ShutDown.BUSY OR ShutDown.ERR OR NOT WritePersistentData.BUSY         				
		THEN                   
			Error											:= WritePersistentData.ERR OR ShutDown.ERR;
			ErrorId											:= SEL(WritePersistentData.ERR, ShutDown.ERRID , WritePersistentData.ERRID);
			IF UpsMode = eSUPS_ImmediateShutdown
			THEN
				status										:= eSUPS_WaitForPowerOFF;
			ELSIF UpsMode = eSUPS_WrPersistData_NoShutdown
			THEN
				status										:= eSUPS_WaitForRecover;
				state										:= 0;
			ELSE //Stop TC and write persistent data
				state										:= state + 1;
			END_IF		
		END_IF                          				
													
	902:(*Tc Stop*)                       	
		TcStop(STOP := TRUE);
		IF NOT TcStop.BUSY
		THEN
			Error											:= Error OR TcStop.ERR;
			ErrorId											:= SEL(TcStop.ERR, ErrorId, TcStop.ERRID);
			status											:= eSUPS_WaitForPowerOFF;
		END_IF
			
	END_CASE

ELSE
	Status													:= eSUPS_PowerOK;
	state													:= 0;
	Error													:= FALSE;
	ErrorID													:= 0;	
	PowerFailDetect											:= FALSE;
END_IF

(********************************************************************)

END_FUNCTION_BLOCK

// ---- POUs/Logging/DataUdpLogger.TcPOU
{attribute 'no_check' := ''}
//Extension to FB "DoubleBuffer" to stream data continuously via UDP, max buffer size is 2 * Tc2_TCP.Param.TCPADS_MAXUDP_BUFFSIZE (2*8192)
{attribute 'enable_dynamic_creation'}
FUNCTION_BLOCK DataUdpLogger EXTENDS DoubleBuffer
VAR_OUTPUT CONSTANT 
{attribute 'displaymode':='binary'}
	OPTION_KEEP_PORT_OPEN_ON_ERROR							: 	BYTE := 2#0000_0001; //Keep file open in error case to be able to contine after reset
{attribute 'displaymode':='binary'}
	OPTION_ADD_DATA_WHEN_DISABLED							:	BYTE := 2#0000_0010; //Allows to add data when disabled
{attribute 'displaymode':='binary'}
	OPTION_ENABLE_DEBUG										:	BYTE := 2#1000_0000; //Creates ADS log entries for conection events and errors
END_VAR                     								
VAR_INPUT                   								
	Enable													: 	BOOL; //Enable to write looked data cyclic into file  
	ResetTrig												: 	BOOL; //Reset internal error 

{attribute 'displaymode':='binary'}
	Options													: 	BYTE := 2#00000000; // See outputs constant OPTION_xxx
	LocalHost	 											: 	T_IPv4Addr;  	//Local (client) address. String containing an (Ipv4) Internet Protocol dotted address. 
	LocalPort												:	UDINT := 515;	//Local (client) Internet Protocol (IP) port. (TCP Port = 1468) *)	
	RemoteHost	 											: 	T_IPv4Addr;  	//Remote (server) address. String containing an (Ipv4) Internet Protocol dotted address. 
	RemotePort												:	UDINT := 514;	//Remote (server) Internet Protocol (IP) port. (TCP Port = 1468) 
END_VAR                     								
VAR_IN_OUT                  								
END_VAR                     								
VAR_OUTPUT       
	TimeSendData											:	TIME; //Elapsed time to send data package 
	CounterSendData											:	UDINT; //Endless counter of packages sent 
	MaxTimeSendData											:	TIME;
	Online													:	BOOL; //TRUE if coonection is sucessful etablished
	hSocket													: 	T_HSOCKET ; //UDP Socket handle
	Busy													: 	BOOL; //Stream data active
	Error													: 	BOOL;       
{attribute 'displaymode':='hex'}
	ErrorId													:	UDINT;	//See Beckhoff TF6310/ADS documentation for more information regarding error code
	ErrorFnc												:	STRING(20); //Error source 
	WinsockErrorId											:	E_WinsockError; //Winsocket error enum - see TF6310 documentation for further information
END_VAR                     								
VAR            
//local ************************************************************************************

	State													: 	INT;
	SendErrorCnt											:	INT;
	StartTimeSendData										:	TIME;			
;

//trigger *********************************************************************************

//timer ***********************************************************************************

//instances ***********************************************************************************             								
	SocketClose												:	FB_SocketClose := (tTimeout := DEFAULT_ADS_TIMEOUT);
	SocketUdpCreate 										:	FB_SocketUdpCreate := (tTimeout := DEFAULT_ADS_TIMEOUT);
	SocketUdpSend											:	FB_SocketUdpSendTo := (tTimeout := T#10S);
	
//Dummys ****************************************************************************************

END_VAR

(* Data logger via UDP stream based on two buffer concept			*)
(********************************************************************)

(* Server connection ************************************************)
	CASE state OF
	0:
		IF Error
		THEN
			IF NOT Enable OR ResetTrig 
			THEN //Reset error
				Error										:= FALSE;
				ErrorId										:= 0;
				ErrorFnc									:= '';	
				WinsockErrorId								:= WSOK;	

				SocketUdpCreate(bExecute := FALSE);
				SocketClose(bExecute := FALSE);
				SocketUdpSend(bExecute := FALSE);		
			END_IF		
		ELSIF Online AND Enable
		THEN	
			IF hr <> S_OK
			THEN //Method executed with error
				Error										:= TRUE;
				ErrorId										:= HRESULT_TO_ADSERROR(hr);
		
			ELSIF ReadyToRead //Buffer full or triggered by interval
			THEN
				StartTimeSendData							:= TIME();

				SocketUdpSend(
					sSrvNetId	:= , 
					hSocket		:= hSocket, 
					sRemoteHost	:= RemoteHost, 
					nRemotePort	:= RemotePort, 
					cbLen		:= SizeOfDataToRead, 
					pSrc		:= pDataToRead, 
					bExecute	:= TRUE, 
					tTimeout	:= , 
					bBusy		=> , 
					bError		=> , 
					nErrId		=> );
													
				state										:= 20;
			END_IF
		ELSIF Enable			
		THEN
			SocketUdpCreate(bExecute := FALSE);
			SocketClose(bExecute := FALSE);
			SocketUdpSend(bExecute := FALSE);
			Online											:= FALSE;
			Busy											:= TRUE;
			Error											:= FALSE;
			ErrorId											:= 0;
			ErrorFnc										:= '';	
			WinsockErrorId									:= WSOK;
			
			IF NOT SocketUdpCreate.bBusy
				AND NOT SocketClose.bBusy
				AND NOT SocketUdpSend.bBusy
			THEN
				SocketUdpCreate(
					sSrvNetId	:= , 
					sLocalHost	:= LocalHost, 
					nLocalPort	:= LocalPort, 
					bExecute	:= TRUE, 
					tTimeout	:= , 
					bBusy		=> , 
					bError		=> , 
					nErrId		=> , 
					hSocket		=> hSocket);
				CounterSendData								:= 0;
				SendErrorCnt								:= 0;
				state										:= 10;
			END_IF	
		ELSE //Disabled
			IF hSocket.handle <> 0
			THEN //Close socket
				IF NOT Empty 
				THEN //Write rest of buffer
					IF NOT ReadyToRead THEN setReadyToRead(TRUE); END_IF 
					StartTimeSendData						:= TIME();
					SocketUdpSend(
						sSrvNetId	:= , 
						hSocket		:= hSocket, 
						sRemoteHost	:= RemoteHost, 
						nRemotePort	:= RemotePort, 
						cbLen		:= SizeOfDataToRead, 
						pSrc		:= pDataToRead, 
						bExecute	:= TRUE, 
						tTimeout	:= , 
						bBusy		=> , 
						bError		=> , 
						nErrId		=> );
					State									:= 20;
				ELSE
					SocketClose(bExecute := hSocket.handle <> 0,  hSocket := hSocket);
					State									:= 30;
				END_IF			
			END_IF
		END_IF

	(* Create Socket *******************************************************)
	10: 
		SocketUdpCreate(
			sSrvNetId	:= , 
			sLocalHost	:= LocalHost, 
			nLocalPort	:= LocalPort, 
			bExecute	:= TRUE, 
			tTimeout	:= , 
			bBusy		=> , 
			bError		=> , 
			nErrId		=> , 
			hSocket		=> hSocket);
			
		IF NOT SocketUdpCreate.bBusy
		THEN
			IF SocketUdpCreate.bError
			THEN
				Error										:= TRUE;
				ErrorId										:= SocketUdpCreate.nErrId;
				ErrorFnc									:= 'SocketUdpCreate';
				WinsockErrorId								:= ADSERROR_TO_WSERROR(ErrorId);
				
				IF Options.7
				THEN
					AdsLogError(CONCAT('LogbookClientSysLog | SocketUdpCreate %s | error id 16#', DWORD_TO_HEXSTR(TO_DWORD(ErrorID),4,FALSE)) ,HSOCKET_TO_STRING(SocketUdpCreate.hSocket));
				END_IF	

				state										:= 30;
			ELSE				
				hSocket.remoteAddr.sAddr					:= RemoteHost;
				hSocket.remoteAddr.nPort					:= RemotePort;
				
				IF Options.7
				THEN
					AdsLogError(CONCAT('LogbookClientSysLog | SocketUdpCreate %s done', '') , HSOCKET_TO_STRING(SocketUdpCreate.hSocket));
				END_IF	
				
				Online 										:= TRUE;
				IF ReadyToRead
				THEN //Write request acitive
					SocketUdpSend(
						sSrvNetId	:= , 
						hSocket		:= hSocket, 
						sRemoteHost	:= RemoteHost, 
						nRemotePort	:= RemotePort, 
						cbLen		:= SizeOfDataToRead, 
						pSrc		:= pDataToRead, 
						bExecute	:= TRUE, 
						tTimeout	:= , 
						bBusy		=> , 
						bError		=> , 
						nErrId		=> );					
					StartTimeSendData						:= TIME();
					State									:= 20;
				ELSE
					State									:= 0;
				END_IF		
				
			END_IF		
			SocketUdpCreate(bExecute:= FALSE);
		END_IF		
		
	(* Send message ****************************************************)
	20:
		SocketUdpSend(
			sSrvNetId	:= , 
			hSocket		:= hSocket, 
			sRemoteHost	:= RemoteHost, 
			nRemotePort	:= RemotePort, 
			cbLen		:= SizeOfDataToRead, 
			pSrc		:= pDataToRead, 
			bExecute	:= TRUE, 
			tTimeout	:= , 
			bBusy		=> , 
			bError		=> , 
			nErrId		=> );
					
		IF NOT SocketUdpSend.bBusy
		THEN
			
			IF SocketUdpSend.bError
			THEN
				IF SendErrorCnt >= 3
				THEN
					Error									:= TRUE;
					ErrorId									:= SocketUdpSend.nErrId;
					ErrorFnc								:= 'SocketUdpSend';
					WinsockErrorId							:= ADSERROR_TO_WSERROR(ErrorId);
	
					IF Options.7
					THEN
						AdsLogError(CONCAT('LogbookClientSysLog | SocketUdpSend %s | error id 16#', DWORD_TO_HEXSTR(TO_DWORD(ErrorID),4,FALSE)) ,HSOCKET_TO_STRING(SocketUdpCreate.hSocket));
					END_IF	
					setReadyToRead(FALSE);
					State									:= 30; //Close socket
				ELSE //Try to send a second time
					SendErrorCnt							:= SendErrorCnt + 1;
				END_IF
			ELSE		
				TimeSendData								:= TIME() - StartTimeSendData;
				MaxTimeSendData								:= MAX(MaxTimeSendData,TimeSendData);
				setReadyToRead(FALSE);
				CounterSendData								:= CounterSendData + 1;		
				SendErrorCnt								:= 0;	
				State										:= SEL(NOT Enable AND Options.1 , 0 ,30);	//Close socket when add data while disabled is allowed, otherwise empty buffer  		
			END_IF 
			
			SocketUdpSend(bExecute := FALSE);
		END_IF
		
	(* Close socket ***********************************************)
	30:	
		SocketClose(
			sSrvNetId	:= , 
			hSocket		:= hSocket, 
			bExecute	:= hSocket.handle <> 0, 
			tTimeout	:= , 
			bBusy		=> , 
			bError		=> , 
			nErrId		=> );

		IF NOT SocketClose.bBusy
		THEN	
			IF SocketClose.bError 
			THEN
				IF NOT Error
				THEN
					Error									:= TRUE;
					ErrorId									:= SocketClose.nErrId;
					ErrorFnc								:= 'SocketUdpClose';
					WinsockErrorId							:= ADSERROR_TO_WSERROR(ErrorId);
				END_IF
				IF Options.7
				THEN
					AdsLogError( CONCAT('LogbookClientSysLog | SocketClose %s | error id 16#', DWORD_TO_HEXSTR(TO_DWORD(ErrorID),4,FALSE)) ,HSOCKET_TO_STRING(SocketClose.hSocket));
				END_IF
				state										:= 0;				
			ELSE    
				IF Options.7
				THEN
					AdsLogError( CONCAT('LogbookClientSysLog | SocketClose %s done', '') , HSOCKET_TO_STRING(SocketClose.hSocket));
				END_IF	
                             
				state										:= 0;
			END_IF		
			Online											:= FALSE;      
			hSocket.handle 									:= 0; 
			SocketClose(bExecute := FALSE);
		END_IF		
			
	END_CASE

(* Status **********************************************************)
	Busy 													:= State <> 0 OR hSocket.handle <> 0 AND NOT Error;
(**************************************************************************)

METHOD PUBLIC addData : HRESULT //Add data into write buffer and swap if if buffer is filled
VAR_INPUT
	pData													:	POINTER TO BYTE;
	SizeofData												:	UDINT;
END_VAR
IF NOT Error AND(Enable OR Options.1)
THEN 
	IF SUPER^.addData(pData,SizeOfData) <> S_OK
	THEN
		ErrorId												:= HRESULT_TO_ADSERROR(hr);
		Error												:= TRUE;
	END_IF
ELSE
	addData													:= SEL(hr <> S_OK , E_HRESULTADSERR.INVALIDACCESS ,hr);
END_IF
END_METHOD

METHOD PUBLIC addString : HRESULT //Add string to write buffer and swap if buffer is filled
VAR_INPUT
	Data													:	T_MAXSTRING;
END_VAR
addString := This^.addData(ADR(Data),TO_UDINT(LEN(Data)));
END_METHOD

PROPERTY PUBLIC optAddDataWhenDisabled : BOOL
GET
optKeepPortOpenOnError := Options.1;
END_GET
SET
Options.1				:= optKeepPortOpenOnError;
END_SET
END_PROPERTY

PROPERTY PUBLIC optEnableAdsErrorLog : BOOL
GET
optEnableAdsErrorLog := Options.7;
END_GET
SET
Options.7				:= optEnableAdsErrorLog;
END_SET
END_PROPERTY

PROPERTY PUBLIC optKeepPortOpenOnError : BOOL
GET
optKeepPortOpenOnError := Options.0;
END_GET
SET
Options.0				:= optKeepPortOpenOnError;
END_SET
END_PROPERTY

//Reset buffer 
METHOD PUBLIC reset : BOOL //TRUE if method is finnished
VAR_INPUT
END_VAR

MaxTimeSendData := T#0MS;
reset := SUPER^.reset();
END_METHOD

END_FUNCTION_BLOCK

// ---- POUs/Motion/TF50xx-NC/02_Options/Parameter/AxPara.TcPOU
{attribute 'no_check'}
//FB to read and write NC axis parameter. 
//The FB can be enherided and derivatived methods of SeqRead/SeqWrite used for application specific parameter.
//The extended methods need to call the super class at the beginning and return true if execution will be finished. The allowed states for new parameter are 1..99
FUNCTION_BLOCK AxPara EXTENDS AxRWParaBase
VAR_OUTPUT CONSTANT
END_VAR                                 					
VAR_INPUT                               					                                   	                                        	
	AxisID													: 	UDINT;				(* ID der Achse *)

	(* zu schreibende Achparameter *)
	SetLimitPosActive										: 	BOOL;
	SetLimitNegActive										:	BOOL;
	SetLimitPos												: 	LREAL;
	SetLimitNeg												: 	LREAL;
                                    						
	SetRefFlag												:	BOOL;
                                    						
	SetTargetPosWindow										:	LREAL;
	SetTargetPosWindowMonitoring							:	BOOL;
	SetPosRangeWindow										: 	LREAL;
	SetPosRangeWindowMonitoring								:	BOOL;

	SetDynamicsRefVelocity									: 	LREAL;
	SetDynamicsMaxVelocity									: 	LREAL;
	SetG0Velocity											: 	LREAL;
	SetRefVelocityPos										: 	LREAL;
	SetRefVelocityNeg										: 	LREAL;
	SetManVelocityFast										: 	LREAL;
	SetManVelocitySlow										: 	LREAL;

	SetKv													: 	LREAL;
	SetJerk													: 	LREAL;
	SetAcc													: 	LREAL;
	SetDec													: 	LREAL;
	SetMaxPosLagValue										: 	LREAL;
	SetMaxPosLagFilterTime									: 	LREAL;
	
	SetMaxPosLagMonitoring									: 	BOOL;
                                        					
	SetModuloFactor 										:	LREAL;
	SetToleranceWindowModuloStart							:	LREAL;
	SetInvertEncCoutingDir									:	BOOL; //UINT;
                                        					
	SetEncScalingNumerator									:	LREAL; //Scaling idx 16#6 replaced by Numerator and Denominator
	SetEncScalingDenominator								:	LREAL; //Scaling idx 16#6 replaced by Numerator and Denominator
	SetPosBias												: 	LREAL; (* NC positon offset *)
	SetReferenceSystem										:	UDINT; //incremental, absolute, abs modulo
	SetCalibrationValue										: 	LREAL;	(* read/write only allowed for certain encoder types *)
	SetCalibrationMode										:	UDINT; 
	SetCalibrInvertDirForCamSearch							:	BOOL; (* TRUE=Cam search direction negative , read/write only allowed for certain encoder types *)
	SetCalibrInvertDirForSyncImpSearch						:	BOOL; (* TRUE=Sync impuls (off cam) search direction negative, read/write only allowed for certain encoder types *)
	
	SetInvertMotorPolarity									: 	BOOL; //UINT;
                                							  	
	SetBreakingDistancePos									: 	LREAL;
	SetBreakingDistanceNeg									: 	LREAL;
END_VAR                                 					
VAR_OUTPUT                              										
	Name													: STRING(30) := '';
	AxisType												: UDINT := 0; (* Nc axis type :
																								0	NOT DEFINED
																								1	Continuous axis (stepper motor)
																								2	Diskrete Achse (Eil/Schleich)
																								3	Continuous axis (stepper motor)
																								5	Encoder axis/ simulation axis 
																								6	NcAxisType_Hydraulic            
																								7	NcAxisType_TimeGenerator       
																								100	NcAxisType_Specific      *)
                                        					
